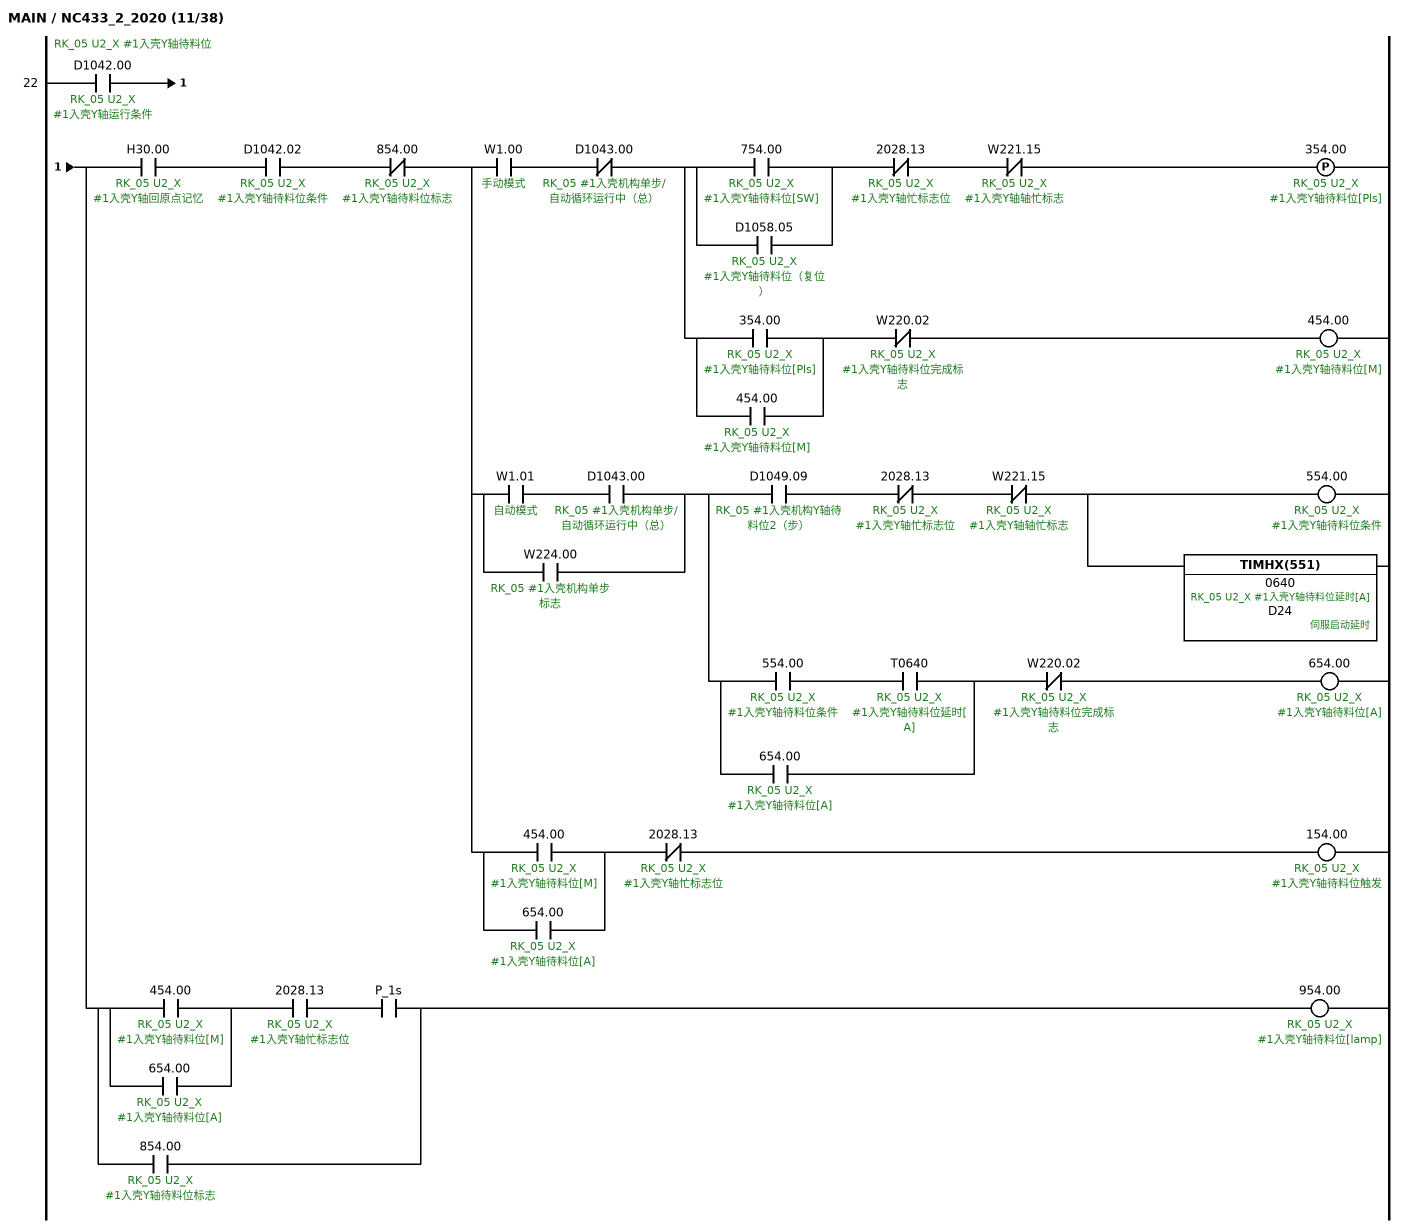
; [picture p120: MAIN / NC433_2_2020, rungs 22-22]
; rung 22: RK_05 U2_X #1入壳Y轴待料位
LD D1042.00  ; RK_05 U2_X #1入壳Y轴运行条件
OUT TR0
AND H30.00  ; RK_05 U2_X #1入壳Y轴回原点记忆
AND D1042.02  ; RK_05 U2_X #1入壳Y轴待料位条件
ANDNOT 854.00  ; RK_05 U2_X #1入壳Y轴待料位标志
OUT TR1
AND W1.00  ; 手动模式
ANDNOT D1043.00  ; RK_05 #1入壳机构单步/自动循环运行中（总）
OUT TR2
LD 754.00  ; RK_05 U2_X #1入壳Y轴待料位[SW]
OR D1058.05  ; RK_05 U2_X #1入壳Y轴待料位（复位）
ANDLD
ANDNOT 2028.13  ; RK_05 U2_X #1入壳Y轴忙标志位
ANDNOT W221.15  ; RK_05 U2_X #1入壳Y轴轴忙标志
DIFU(013) 354.00  ; RK_05 U2_X #1入壳Y轴待料位[Pls]
LD TR2
LD 354.00  ; RK_05 U2_X #1入壳Y轴待料位[Pls]
OR 454.00  ; RK_05 U2_X #1入壳Y轴待料位[M]
ANDLD
ANDNOT W220.02  ; RK_05 U2_X #1入壳Y轴待料位完成标志
OUT 454.00  ; RK_05 U2_X #1入壳Y轴待料位[M]
LD TR1
LD W1.01  ; 自动模式
AND D1043.00  ; RK_05 #1入壳机构单步/自动循环运行中（总）
OR W224.00  ; RK_05 #1入壳机构单步标志
ANDLD
OUT TR2
AND D1049.09  ; RK_05 #1入壳机构Y轴待料位2（步）
ANDNOT 2028.13  ; RK_05 U2_X #1入壳Y轴忙标志位
ANDNOT W221.15  ; RK_05 U2_X #1入壳Y轴轴忙标志
OUT 554.00  ; RK_05 U2_X #1入壳Y轴待料位条件
TIMHX(551) 0640 D24  ; 伺服启动延时, RK_05 U2_X #1入壳Y轴待料位延时[A]
LD TR2
LD 554.00  ; RK_05 U2_X #1入壳Y轴待料位条件
AND T0640  ; RK_05 U2_X #1入壳Y轴待料位延时[A]
OR 654.00  ; RK_05 U2_X #1入壳Y轴待料位[A]
ANDLD
ANDNOT W220.02  ; RK_05 U2_X #1入壳Y轴待料位完成标志
OUT 654.00  ; RK_05 U2_X #1入壳Y轴待料位[A]
LD TR1
LD 454.00  ; RK_05 U2_X #1入壳Y轴待料位[M]
OR 654.00  ; RK_05 U2_X #1入壳Y轴待料位[A]
ANDLD
ANDNOT 2028.13  ; RK_05 U2_X #1入壳Y轴忙标志位
OUT 154.00  ; RK_05 U2_X #1入壳Y轴待料位触发
LD TR0
LD 454.00  ; RK_05 U2_X #1入壳Y轴待料位[M]
OR 654.00  ; RK_05 U2_X #1入壳Y轴待料位[A]
AND 2028.13  ; RK_05 U2_X #1入壳Y轴忙标志位
AND P_1s
OR 854.00  ; RK_05 U2_X #1入壳Y轴待料位标志
ANDLD
OUT 954.00  ; RK_05 U2_X #1入壳Y轴待料位[lamp]

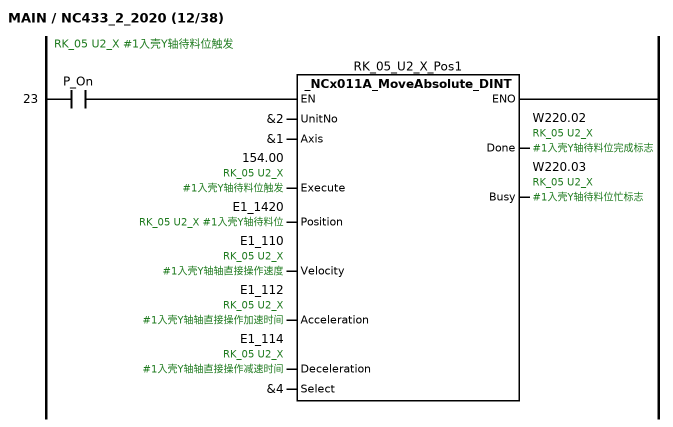
; rung 23: RK_05 U2_X #1入壳Y轴待料位触发
LD P_On
CALL RK_05_U2_X_Pos1 : _NCx011A_MoveAbsolute_DINT (UnitNo := &2, Axis := &1, Execute := 154.00, Position := E1_1420, Velocity := E1_110, Acceleration := E1_112, Deceleration := E1_114, Select := &4, Done => W220.02, Busy => W220.03)  ; RK_05 U2_X #1入壳Y轴待料位触发, RK_05 U2_X #1入壳Y轴待料位, RK_05 U2_X #1入壳Y轴轴直接操作速度, RK_05 U2_X #1入壳Y轴轴直接操作加速时间, RK_05 U2_X #1入壳Y轴轴直接操作减速时间, RK_05 U2_X #1入壳Y轴待料位完成标志, RK_05 U2_X #1入壳Y轴待料位忙标志

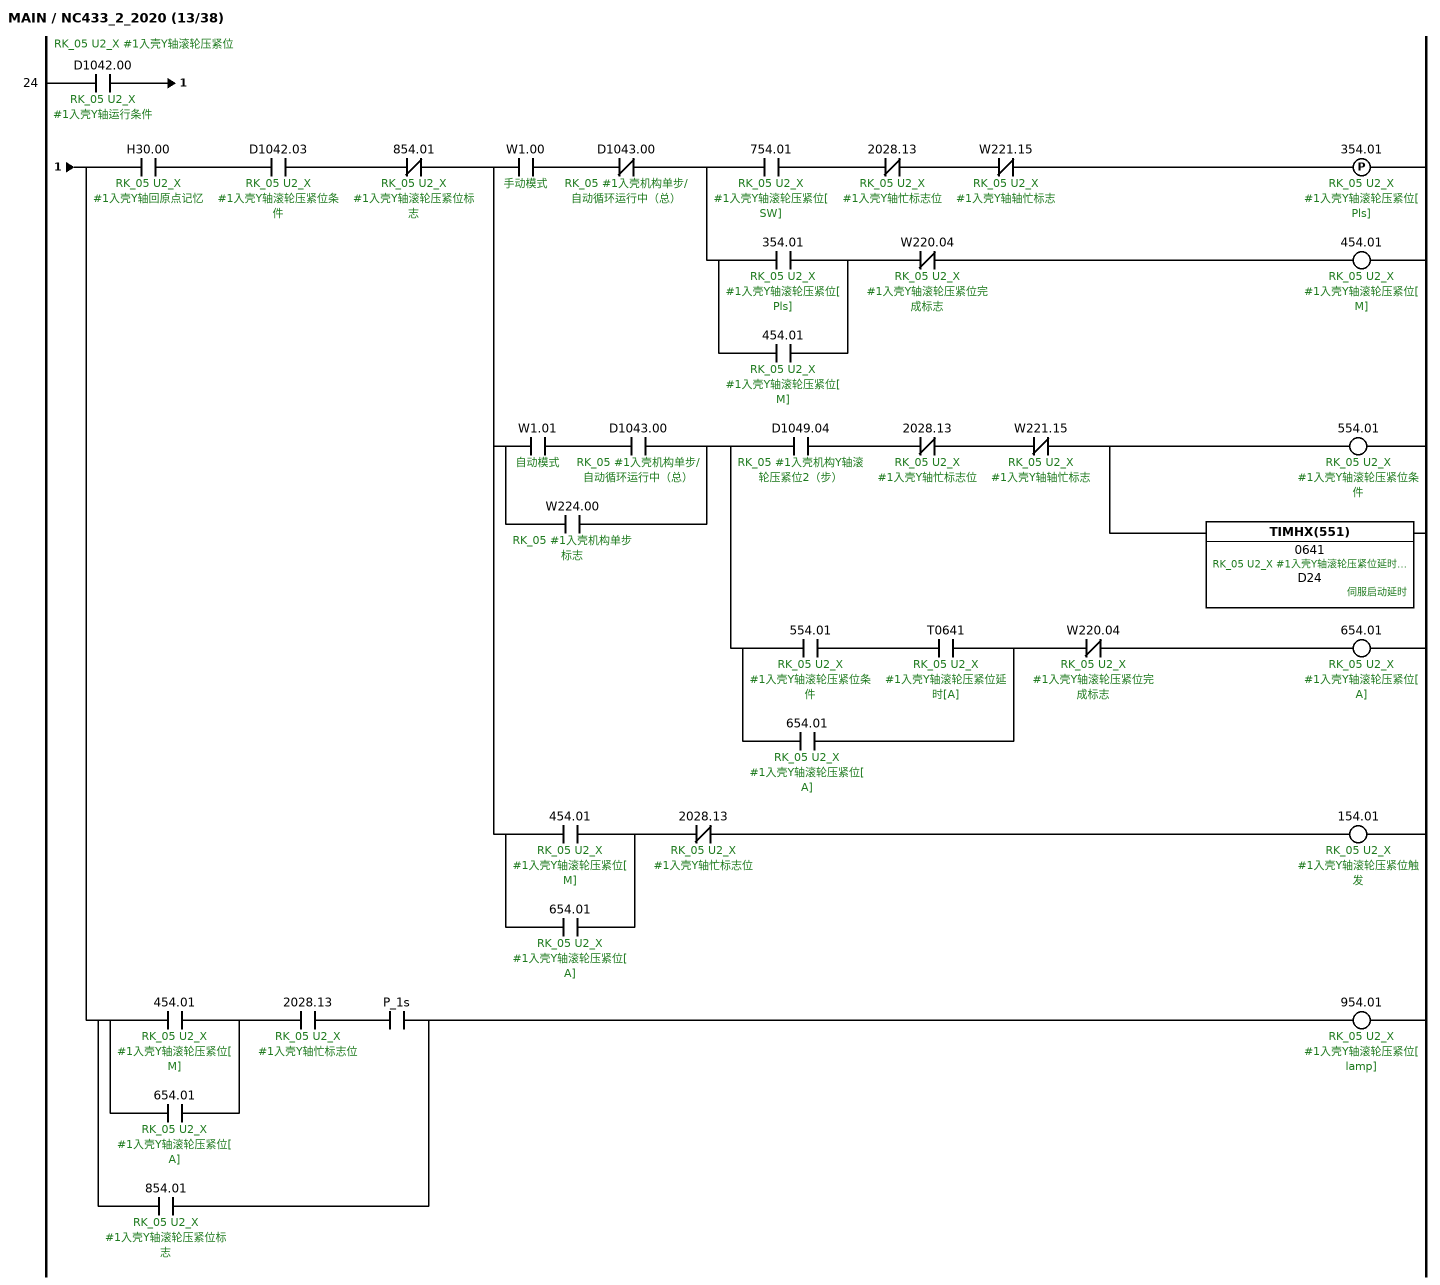
; rung 24: RK_05 U2_X #1入壳Y轴滚轮压紧位
LD D1042.00  ; RK_05 U2_X #1入壳Y轴运行条件
OUT TR0
AND H30.00  ; RK_05 U2_X #1入壳Y轴回原点记忆
AND D1042.03  ; RK_05 U2_X #1入壳Y轴滚轮压紧位条件
ANDNOT 854.01  ; RK_05 U2_X #1入壳Y轴滚轮压紧位标志
OUT TR1
AND W1.00  ; 手动模式
ANDNOT D1043.00  ; RK_05 #1入壳机构单步/自动循环运行中（总）
OUT TR2
AND 754.01  ; RK_05 U2_X #1入壳Y轴滚轮压紧位[SW]
ANDNOT 2028.13  ; RK_05 U2_X #1入壳Y轴忙标志位
ANDNOT W221.15  ; RK_05 U2_X #1入壳Y轴轴忙标志
DIFU(013) 354.01  ; RK_05 U2_X #1入壳Y轴滚轮压紧位[Pls]
LD TR2
LD 354.01  ; RK_05 U2_X #1入壳Y轴滚轮压紧位[Pls]
OR 454.01  ; RK_05 U2_X #1入壳Y轴滚轮压紧位[M]
ANDLD
ANDNOT W220.04  ; RK_05 U2_X #1入壳Y轴滚轮压紧位完成标志
OUT 454.01  ; RK_05 U2_X #1入壳Y轴滚轮压紧位[M]
LD TR1
LD W1.01  ; 自动模式
AND D1043.00  ; RK_05 #1入壳机构单步/自动循环运行中（总）
OR W224.00  ; RK_05 #1入壳机构单步标志
ANDLD
OUT TR2
AND D1049.04  ; RK_05 #1入壳机构Y轴滚轮压紧位2（步）
ANDNOT 2028.13  ; RK_05 U2_X #1入壳Y轴忙标志位
ANDNOT W221.15  ; RK_05 U2_X #1入壳Y轴轴忙标志
OUT 554.01  ; RK_05 U2_X #1入壳Y轴滚轮压紧位条件
TIMHX(551) 0641 D24  ; 伺服启动延时, RK_05 U2_X #1入壳Y轴滚轮压紧位延时[A]
LD TR2
LD 554.01  ; RK_05 U2_X #1入壳Y轴滚轮压紧位条件
AND T0641  ; RK_05 U2_X #1入壳Y轴滚轮压紧位延时[A]
OR 654.01  ; RK_05 U2_X #1入壳Y轴滚轮压紧位[A]
ANDLD
ANDNOT W220.04  ; RK_05 U2_X #1入壳Y轴滚轮压紧位完成标志
OUT 654.01  ; RK_05 U2_X #1入壳Y轴滚轮压紧位[A]
LD TR1
LD 454.01  ; RK_05 U2_X #1入壳Y轴滚轮压紧位[M]
OR 654.01  ; RK_05 U2_X #1入壳Y轴滚轮压紧位[A]
ANDLD
ANDNOT 2028.13  ; RK_05 U2_X #1入壳Y轴忙标志位
OUT 154.01  ; RK_05 U2_X #1入壳Y轴滚轮压紧位触发
LD TR0
LD 454.01  ; RK_05 U2_X #1入壳Y轴滚轮压紧位[M]
OR 654.01  ; RK_05 U2_X #1入壳Y轴滚轮压紧位[A]
AND 2028.13  ; RK_05 U2_X #1入壳Y轴忙标志位
AND P_1s
OR 854.01  ; RK_05 U2_X #1入壳Y轴滚轮压紧位标志
ANDLD
OUT 954.01  ; RK_05 U2_X #1入壳Y轴滚轮压紧位[lamp]

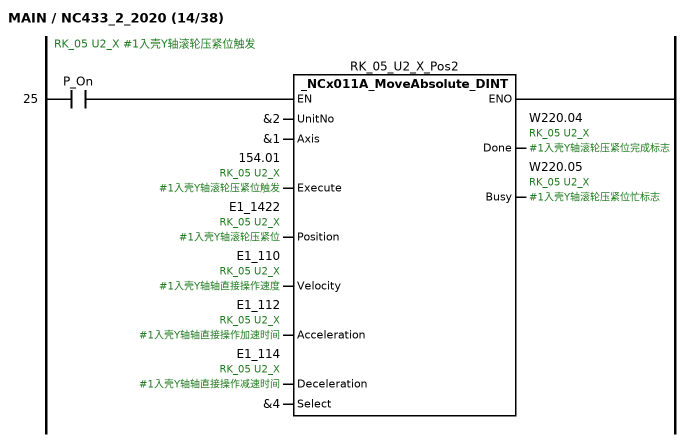
; rung 25: RK_05 U2_X #1入壳Y轴滚轮压紧位触发
LD P_On
CALL RK_05_U2_X_Pos2 : _NCx011A_MoveAbsolute_DINT (UnitNo := &2, Axis := &1, Execute := 154.01, Position := E1_1422, Velocity := E1_110, Acceleration := E1_112, Deceleration := E1_114, Select := &4, Done => W220.04, Busy => W220.05)  ; RK_05 U2_X #1入壳Y轴滚轮压紧位触发, RK_05 U2_X #1入壳Y轴滚轮压紧位, RK_05 U2_X #1入壳Y轴轴直接操作速度, RK_05 U2_X #1入壳Y轴轴直接操作加速时间, RK_05 U2_X #1入壳Y轴轴直接操作减速时间, RK_05 U2_X #1入壳Y轴滚轮压紧位完成标志, RK_05 U2_X #1入壳Y轴滚轮压紧位忙标志

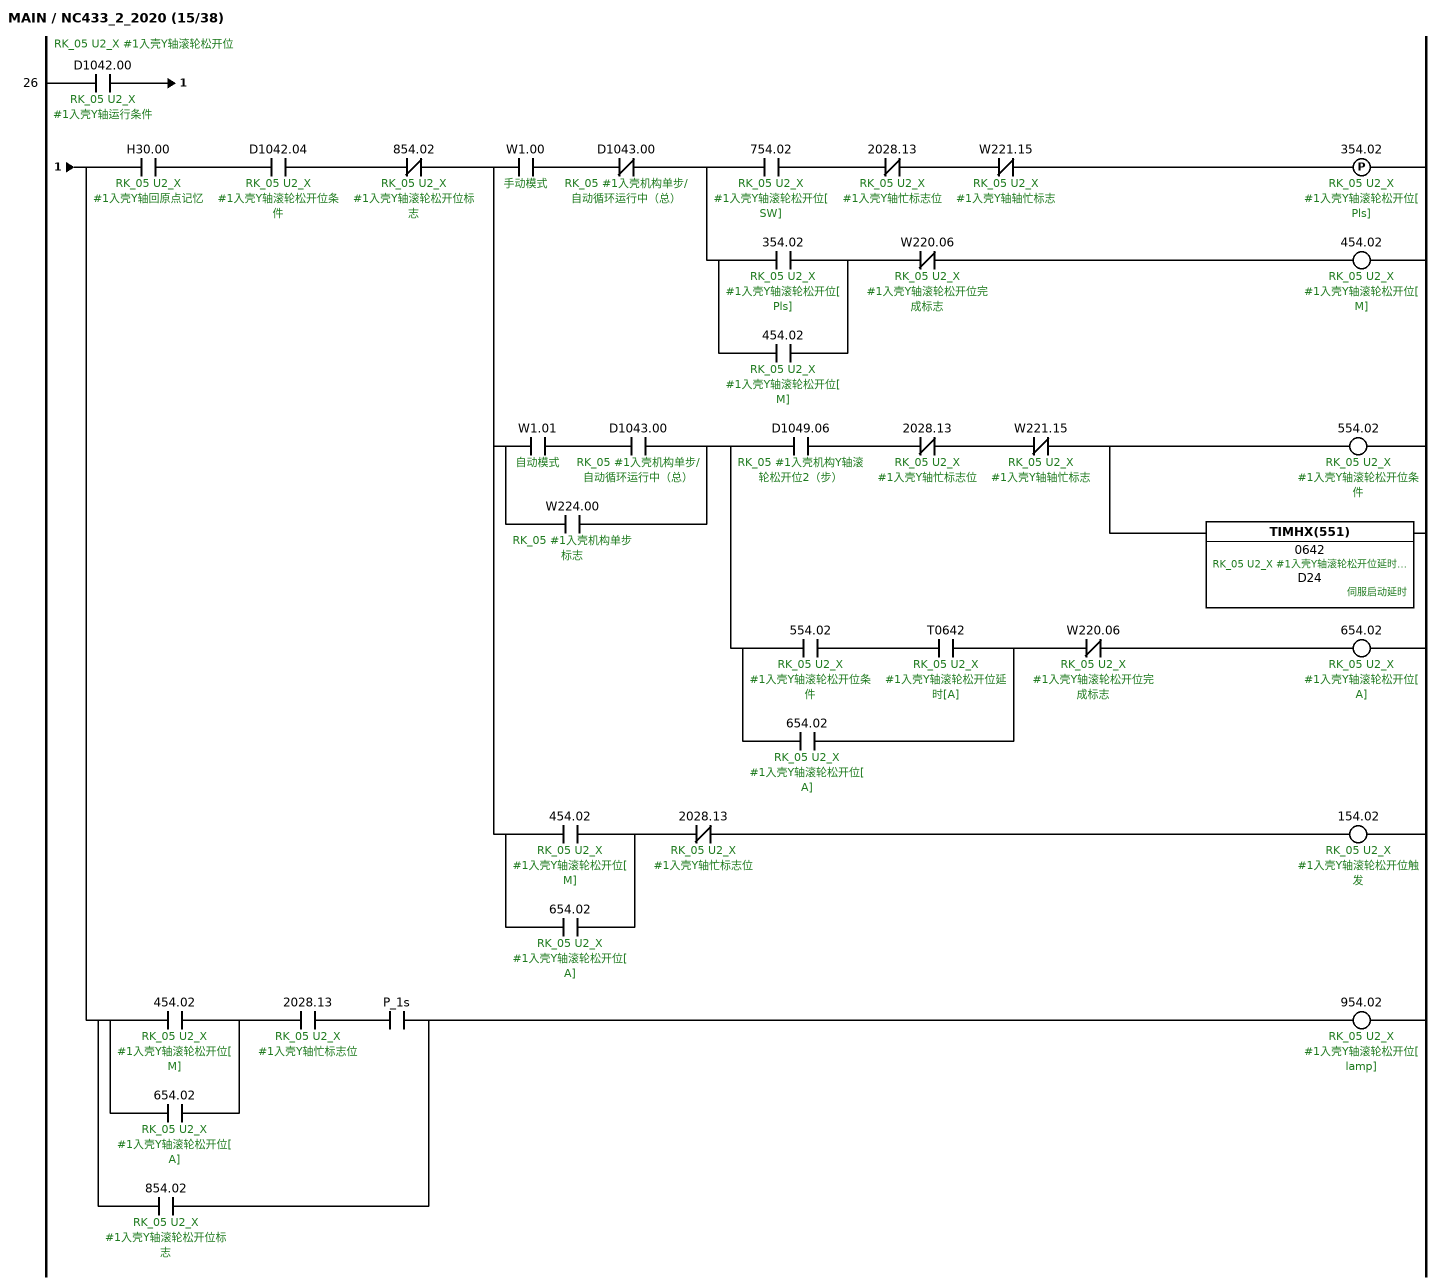
; rung 26: RK_05 U2_X #1入壳Y轴滚轮松开位
LD D1042.00  ; RK_05 U2_X #1入壳Y轴运行条件
OUT TR0
AND H30.00  ; RK_05 U2_X #1入壳Y轴回原点记忆
AND D1042.04  ; RK_05 U2_X #1入壳Y轴滚轮松开位条件
ANDNOT 854.02  ; RK_05 U2_X #1入壳Y轴滚轮松开位标志
OUT TR1
AND W1.00  ; 手动模式
ANDNOT D1043.00  ; RK_05 #1入壳机构单步/自动循环运行中（总）
OUT TR2
AND 754.02  ; RK_05 U2_X #1入壳Y轴滚轮松开位[SW]
ANDNOT 2028.13  ; RK_05 U2_X #1入壳Y轴忙标志位
ANDNOT W221.15  ; RK_05 U2_X #1入壳Y轴轴忙标志
DIFU(013) 354.02  ; RK_05 U2_X #1入壳Y轴滚轮松开位[Pls]
LD TR2
LD 354.02  ; RK_05 U2_X #1入壳Y轴滚轮松开位[Pls]
OR 454.02  ; RK_05 U2_X #1入壳Y轴滚轮松开位[M]
ANDLD
ANDNOT W220.06  ; RK_05 U2_X #1入壳Y轴滚轮松开位完成标志
OUT 454.02  ; RK_05 U2_X #1入壳Y轴滚轮松开位[M]
LD TR1
LD W1.01  ; 自动模式
AND D1043.00  ; RK_05 #1入壳机构单步/自动循环运行中（总）
OR W224.00  ; RK_05 #1入壳机构单步标志
ANDLD
OUT TR2
AND D1049.06  ; RK_05 #1入壳机构Y轴滚轮松开位2（步）
ANDNOT 2028.13  ; RK_05 U2_X #1入壳Y轴忙标志位
ANDNOT W221.15  ; RK_05 U2_X #1入壳Y轴轴忙标志
OUT 554.02  ; RK_05 U2_X #1入壳Y轴滚轮松开位条件
TIMHX(551) 0642 D24  ; 伺服启动延时, RK_05 U2_X #1入壳Y轴滚轮松开位延时[A]
LD TR2
LD 554.02  ; RK_05 U2_X #1入壳Y轴滚轮松开位条件
AND T0642  ; RK_05 U2_X #1入壳Y轴滚轮松开位延时[A]
OR 654.02  ; RK_05 U2_X #1入壳Y轴滚轮松开位[A]
ANDLD
ANDNOT W220.06  ; RK_05 U2_X #1入壳Y轴滚轮松开位完成标志
OUT 654.02  ; RK_05 U2_X #1入壳Y轴滚轮松开位[A]
LD TR1
LD 454.02  ; RK_05 U2_X #1入壳Y轴滚轮松开位[M]
OR 654.02  ; RK_05 U2_X #1入壳Y轴滚轮松开位[A]
ANDLD
ANDNOT 2028.13  ; RK_05 U2_X #1入壳Y轴忙标志位
OUT 154.02  ; RK_05 U2_X #1入壳Y轴滚轮松开位触发
LD TR0
LD 454.02  ; RK_05 U2_X #1入壳Y轴滚轮松开位[M]
OR 654.02  ; RK_05 U2_X #1入壳Y轴滚轮松开位[A]
AND 2028.13  ; RK_05 U2_X #1入壳Y轴忙标志位
AND P_1s
OR 854.02  ; RK_05 U2_X #1入壳Y轴滚轮松开位标志
ANDLD
OUT 954.02  ; RK_05 U2_X #1入壳Y轴滚轮松开位[lamp]

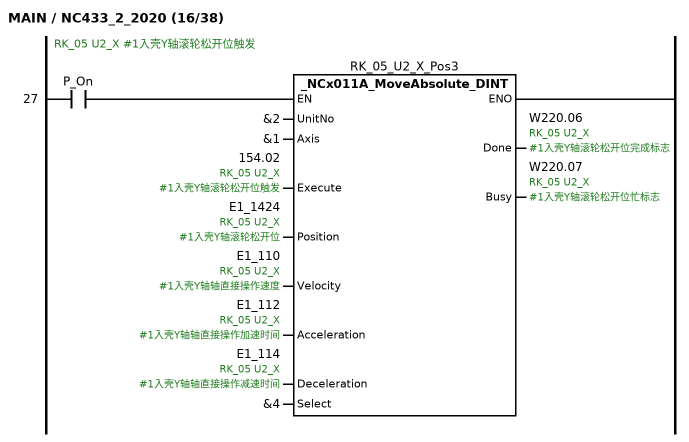
; rung 27: RK_05 U2_X #1入壳Y轴滚轮松开位触发
LD P_On
CALL RK_05_U2_X_Pos3 : _NCx011A_MoveAbsolute_DINT (UnitNo := &2, Axis := &1, Execute := 154.02, Position := E1_1424, Velocity := E1_110, Acceleration := E1_112, Deceleration := E1_114, Select := &4, Done => W220.06, Busy => W220.07)  ; RK_05 U2_X #1入壳Y轴滚轮松开位触发, RK_05 U2_X #1入壳Y轴滚轮松开位, RK_05 U2_X #1入壳Y轴轴直接操作速度, RK_05 U2_X #1入壳Y轴轴直接操作加速时间, RK_05 U2_X #1入壳Y轴轴直接操作减速时间, RK_05 U2_X #1入壳Y轴滚轮松开位完成标志, RK_05 U2_X #1入壳Y轴滚轮松开位忙标志

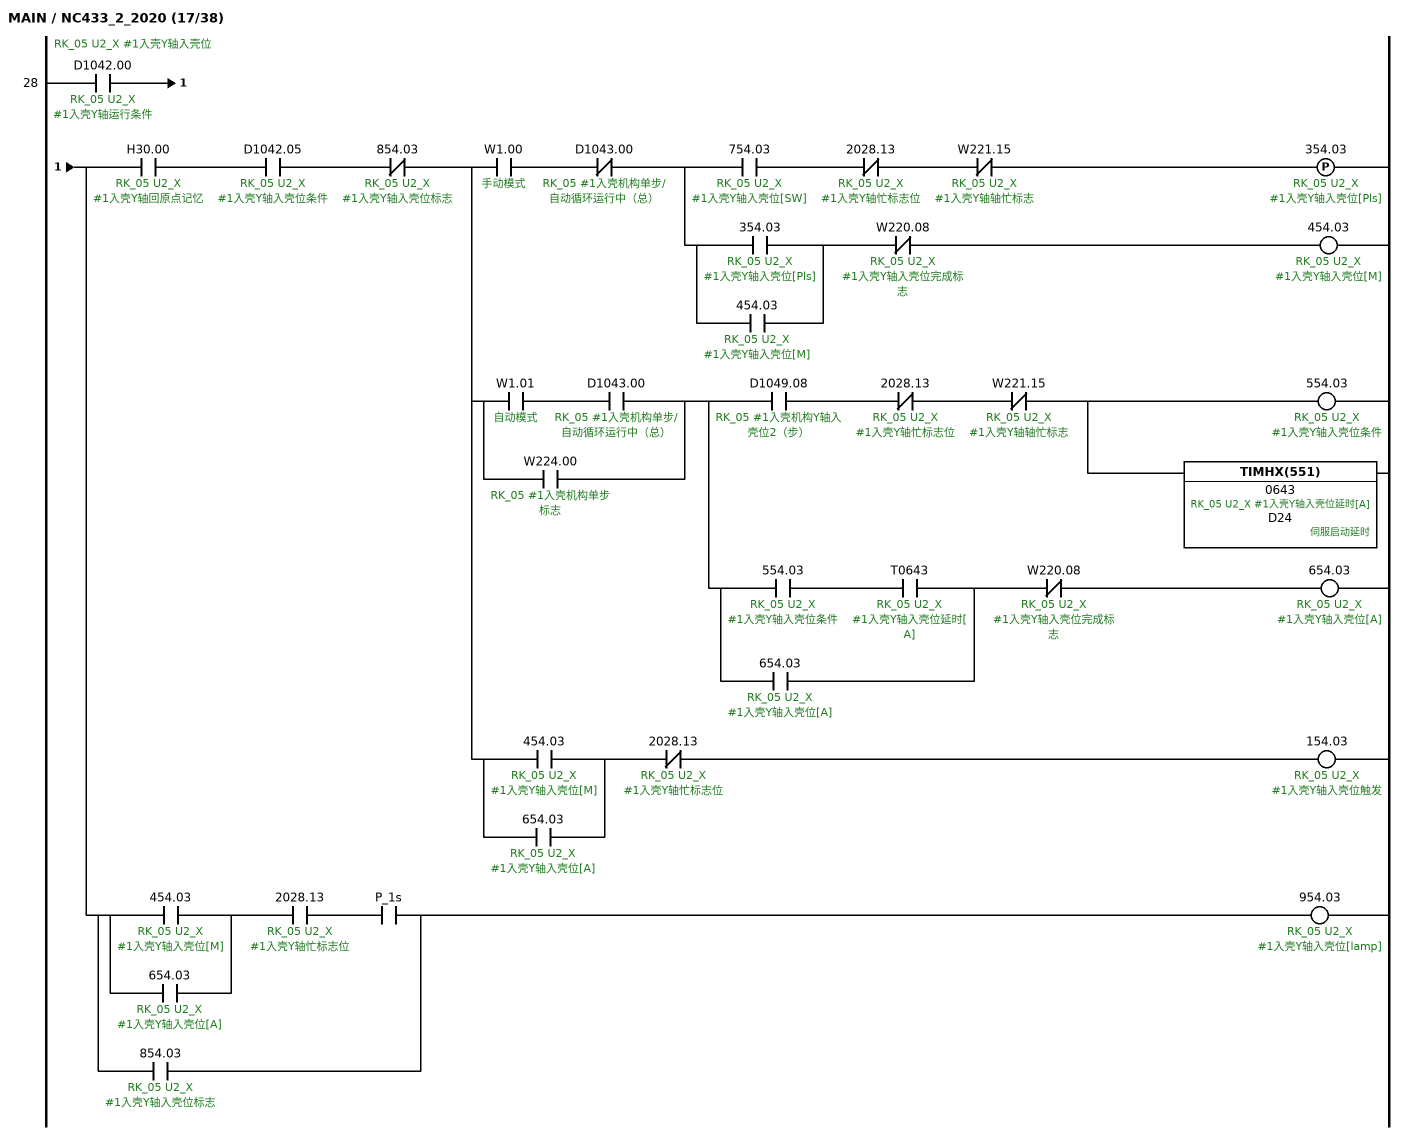
; rung 28: RK_05 U2_X #1入壳Y轴入壳位
LD D1042.00  ; RK_05 U2_X #1入壳Y轴运行条件
OUT TR0
AND H30.00  ; RK_05 U2_X #1入壳Y轴回原点记忆
AND D1042.05  ; RK_05 U2_X #1入壳Y轴入壳位条件
ANDNOT 854.03  ; RK_05 U2_X #1入壳Y轴入壳位标志
OUT TR1
AND W1.00  ; 手动模式
ANDNOT D1043.00  ; RK_05 #1入壳机构单步/自动循环运行中（总）
OUT TR2
AND 754.03  ; RK_05 U2_X #1入壳Y轴入壳位[SW]
ANDNOT 2028.13  ; RK_05 U2_X #1入壳Y轴忙标志位
ANDNOT W221.15  ; RK_05 U2_X #1入壳Y轴轴忙标志
DIFU(013) 354.03  ; RK_05 U2_X #1入壳Y轴入壳位[Pls]
LD TR2
LD 354.03  ; RK_05 U2_X #1入壳Y轴入壳位[Pls]
OR 454.03  ; RK_05 U2_X #1入壳Y轴入壳位[M]
ANDLD
ANDNOT W220.08  ; RK_05 U2_X #1入壳Y轴入壳位完成标志
OUT 454.03  ; RK_05 U2_X #1入壳Y轴入壳位[M]
LD TR1
LD W1.01  ; 自动模式
AND D1043.00  ; RK_05 #1入壳机构单步/自动循环运行中（总）
OR W224.00  ; RK_05 #1入壳机构单步标志
ANDLD
OUT TR2
AND D1049.08  ; RK_05 #1入壳机构Y轴入壳位2（步）
ANDNOT 2028.13  ; RK_05 U2_X #1入壳Y轴忙标志位
ANDNOT W221.15  ; RK_05 U2_X #1入壳Y轴轴忙标志
OUT 554.03  ; RK_05 U2_X #1入壳Y轴入壳位条件
TIMHX(551) 0643 D24  ; 伺服启动延时, RK_05 U2_X #1入壳Y轴入壳位延时[A]
LD TR2
LD 554.03  ; RK_05 U2_X #1入壳Y轴入壳位条件
AND T0643  ; RK_05 U2_X #1入壳Y轴入壳位延时[A]
OR 654.03  ; RK_05 U2_X #1入壳Y轴入壳位[A]
ANDLD
ANDNOT W220.08  ; RK_05 U2_X #1入壳Y轴入壳位完成标志
OUT 654.03  ; RK_05 U2_X #1入壳Y轴入壳位[A]
LD TR1
LD 454.03  ; RK_05 U2_X #1入壳Y轴入壳位[M]
OR 654.03  ; RK_05 U2_X #1入壳Y轴入壳位[A]
ANDLD
ANDNOT 2028.13  ; RK_05 U2_X #1入壳Y轴忙标志位
OUT 154.03  ; RK_05 U2_X #1入壳Y轴入壳位触发
LD TR0
LD 454.03  ; RK_05 U2_X #1入壳Y轴入壳位[M]
OR 654.03  ; RK_05 U2_X #1入壳Y轴入壳位[A]
AND 2028.13  ; RK_05 U2_X #1入壳Y轴忙标志位
AND P_1s
OR 854.03  ; RK_05 U2_X #1入壳Y轴入壳位标志
ANDLD
OUT 954.03  ; RK_05 U2_X #1入壳Y轴入壳位[lamp]

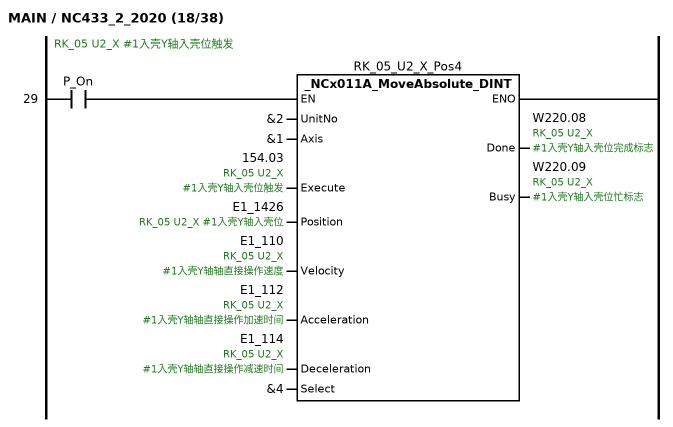
; rung 29: RK_05 U2_X #1入壳Y轴入壳位触发
LD P_On
CALL RK_05_U2_X_Pos4 : _NCx011A_MoveAbsolute_DINT (UnitNo := &2, Axis := &1, Execute := 154.03, Position := E1_1426, Velocity := E1_110, Acceleration := E1_112, Deceleration := E1_114, Select := &4, Done => W220.08, Busy => W220.09)  ; RK_05 U2_X #1入壳Y轴入壳位触发, RK_05 U2_X #1入壳Y轴入壳位, RK_05 U2_X #1入壳Y轴轴直接操作速度, RK_05 U2_X #1入壳Y轴轴直接操作加速时间, RK_05 U2_X #1入壳Y轴轴直接操作减速时间, RK_05 U2_X #1入壳Y轴入壳位完成标志, RK_05 U2_X #1入壳Y轴入壳位忙标志

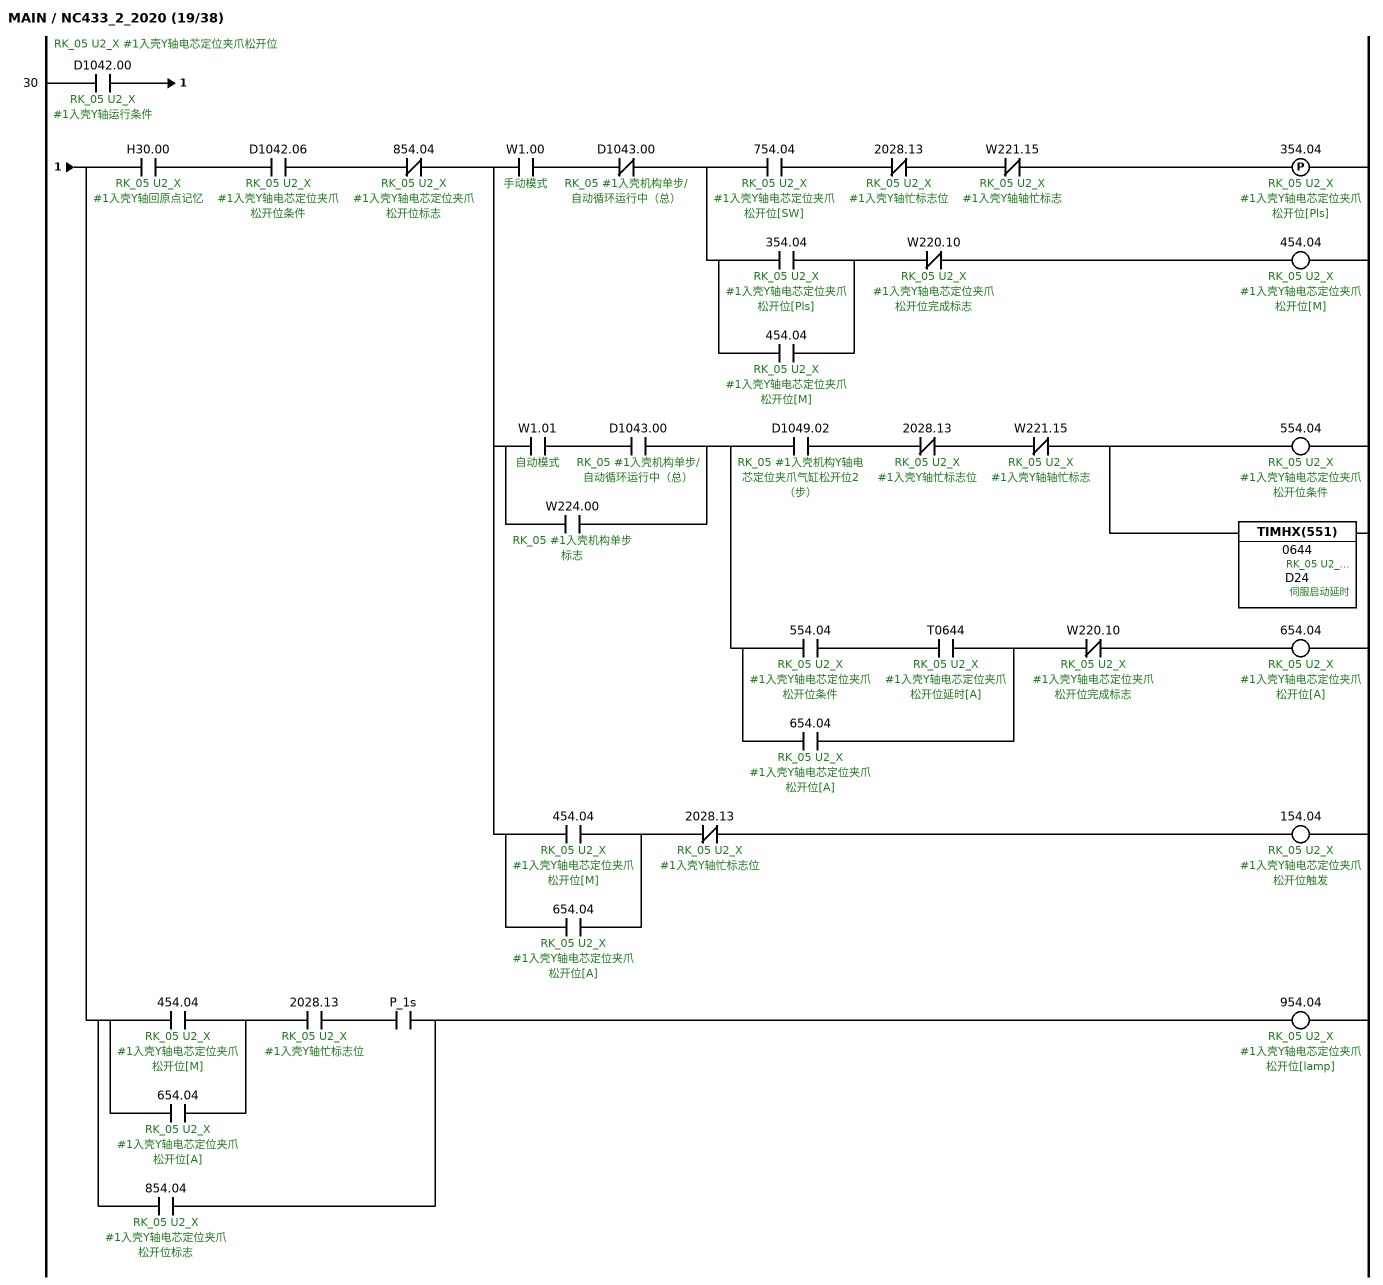
; rung 30: RK_05 U2_X #1入壳Y轴电芯定位夹爪松开位
LD D1042.00  ; RK_05 U2_X #1入壳Y轴运行条件
OUT TR0
AND H30.00  ; RK_05 U2_X #1入壳Y轴回原点记忆
AND D1042.06  ; RK_05 U2_X #1入壳Y轴电芯定位夹爪松开位条件
ANDNOT 854.04  ; RK_05 U2_X #1入壳Y轴电芯定位夹爪松开位标志
OUT TR1
AND W1.00  ; 手动模式
ANDNOT D1043.00  ; RK_05 #1入壳机构单步/自动循环运行中（总）
OUT TR2
AND 754.04  ; RK_05 U2_X #1入壳Y轴电芯定位夹爪松开位[SW]
ANDNOT 2028.13  ; RK_05 U2_X #1入壳Y轴忙标志位
ANDNOT W221.15  ; RK_05 U2_X #1入壳Y轴轴忙标志
DIFU(013) 354.04  ; RK_05 U2_X #1入壳Y轴电芯定位夹爪松开位[Pls]
LD TR2
LD 354.04  ; RK_05 U2_X #1入壳Y轴电芯定位夹爪松开位[Pls]
OR 454.04  ; RK_05 U2_X #1入壳Y轴电芯定位夹爪松开位[M]
ANDLD
ANDNOT W220.10  ; RK_05 U2_X #1入壳Y轴电芯定位夹爪松开位完成标志
OUT 454.04  ; RK_05 U2_X #1入壳Y轴电芯定位夹爪松开位[M]
LD TR1
LD W1.01  ; 自动模式
AND D1043.00  ; RK_05 #1入壳机构单步/自动循环运行中（总）
OR W224.00  ; RK_05 #1入壳机构单步标志
ANDLD
OUT TR2
AND D1049.02  ; RK_05 #1入壳机构Y轴电芯定位夹爪气缸松开位2（步）
ANDNOT 2028.13  ; RK_05 U2_X #1入壳Y轴忙标志位
ANDNOT W221.15  ; RK_05 U2_X #1入壳Y轴轴忙标志
OUT 554.04  ; RK_05 U2_X #1入壳Y轴电芯定位夹爪松开位条件
TIMHX(551) 0644 D24  ; 伺服启动延时, RK_05 U2_X #1入壳Y轴电芯定位夹爪松开位延时[A]
LD TR2
LD 554.04  ; RK_05 U2_X #1入壳Y轴电芯定位夹爪松开位条件
AND T0644  ; RK_05 U2_X #1入壳Y轴电芯定位夹爪松开位延时[A]
OR 654.04  ; RK_05 U2_X #1入壳Y轴电芯定位夹爪松开位[A]
ANDLD
ANDNOT W220.10  ; RK_05 U2_X #1入壳Y轴电芯定位夹爪松开位完成标志
OUT 654.04  ; RK_05 U2_X #1入壳Y轴电芯定位夹爪松开位[A]
LD TR1
LD 454.04  ; RK_05 U2_X #1入壳Y轴电芯定位夹爪松开位[M]
OR 654.04  ; RK_05 U2_X #1入壳Y轴电芯定位夹爪松开位[A]
ANDLD
ANDNOT 2028.13  ; RK_05 U2_X #1入壳Y轴忙标志位
OUT 154.04  ; RK_05 U2_X #1入壳Y轴电芯定位夹爪松开位触发
LD TR0
LD 454.04  ; RK_05 U2_X #1入壳Y轴电芯定位夹爪松开位[M]
OR 654.04  ; RK_05 U2_X #1入壳Y轴电芯定位夹爪松开位[A]
AND 2028.13  ; RK_05 U2_X #1入壳Y轴忙标志位
AND P_1s
OR 854.04  ; RK_05 U2_X #1入壳Y轴电芯定位夹爪松开位标志
ANDLD
OUT 954.04  ; RK_05 U2_X #1入壳Y轴电芯定位夹爪松开位[lamp]

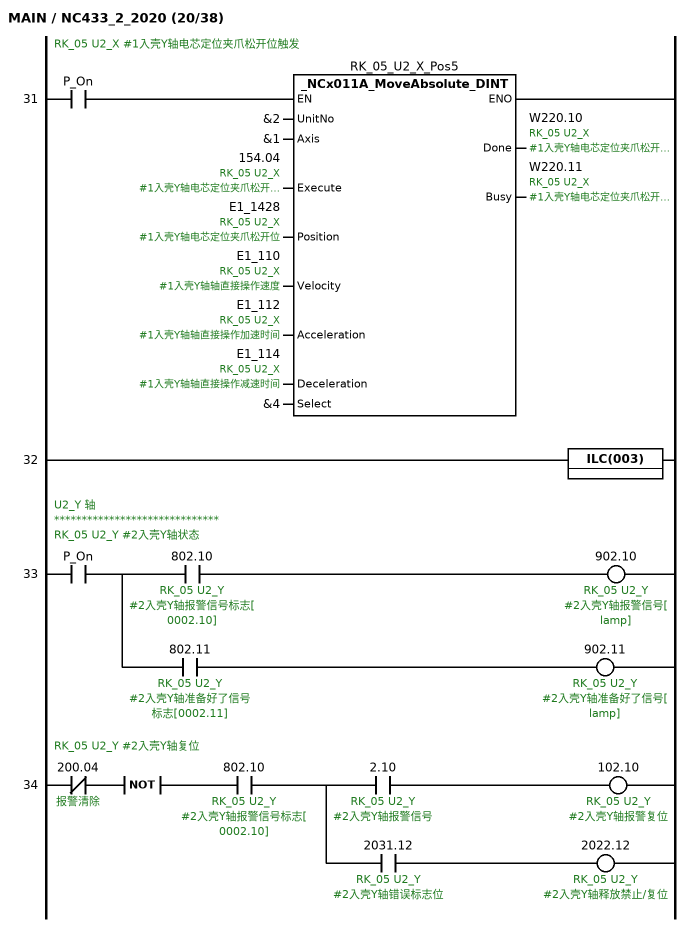
; rung 31: RK_05 U2_X #1入壳Y轴电芯定位夹爪松开位触发
LD P_On
CALL RK_05_U2_X_Pos5 : _NCx011A_MoveAbsolute_DINT (UnitNo := &2, Axis := &1, Execute := 154.04, Position := E1_1428, Velocity := E1_110, Acceleration := E1_112, Deceleration := E1_114, Select := &4, Done => W220.10, Busy => W220.11)  ; RK_05 U2_X #1入壳Y轴电芯定位夹爪松开位触发, RK_05 U2_X #1入壳Y轴电芯定位夹爪松开位, RK_05 U2_X #1入壳Y轴轴直接操作速度, RK_05 U2_X #1入壳Y轴轴直接操作加速时间, RK_05 U2_X #1入壳Y轴轴直接操作减速时间, RK_05 U2_X #1入壳Y轴电芯定位夹爪松开位完成标志, RK_05 U2_X #1入壳Y轴电芯定位夹爪松开位忙标志
; rung 32
ILC(003)
; rung 33: U2_Y 轴 / ****************************** / RK_05 U2_Y #2入壳Y轴状态
LD P_On
OUT TR0
AND 802.10  ; RK_05 U2_Y #2入壳Y轴报警信号标志[0002.10]
OUT 902.10  ; RK_05 U2_Y #2入壳Y轴报警信号[lamp]
LD TR0
AND 802.11  ; RK_05 U2_Y #2入壳Y轴准备好了信号标志[0002.11]
OUT 902.11  ; RK_05 U2_Y #2入壳Y轴准备好了信号[lamp]
; rung 34: RK_05 U2_Y #2入壳Y轴复位
LDNOT 200.04  ; 报警清除
NOT(520)
AND 802.10  ; RK_05 U2_Y #2入壳Y轴报警信号标志[0002.10]
OUT TR0
AND 2.10  ; RK_05 U2_Y #2入壳Y轴报警信号
OUT 102.10  ; RK_05 U2_Y #2入壳Y轴报警复位
LD TR0
AND 2031.12  ; RK_05 U2_Y #2入壳Y轴错误标志位
OUT 2022.12  ; RK_05 U2_Y #2入壳Y轴释放禁止/复位

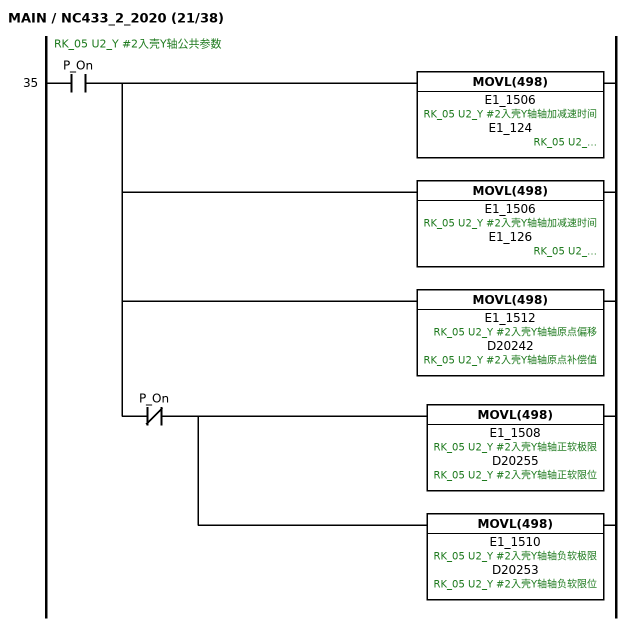
; rung 35: RK_05 U2_Y #2入壳Y轴公共参数
LD P_On
MOVL(498) E1_1506 E1_124  ; RK_05 U2_Y #2入壳Y轴轴加减速时间, RK_05 U2_Y #2入壳Y轴轴直接操作加速时间
MOVL(498) E1_1506 E1_126  ; RK_05 U2_Y #2入壳Y轴轴加减速时间, RK_05 U2_Y #2入壳Y轴轴直接操作减速时间
MOVL(498) E1_1512 D20242  ; RK_05 U2_Y #2入壳Y轴轴原点偏移, RK_05 U2_Y #2入壳Y轴轴原点补偿值
ANDNOT P_On
MOVL(498) E1_1508 D20255  ; RK_05 U2_Y #2入壳Y轴轴正软极限, RK_05 U2_Y #2入壳Y轴轴正软限位
MOVL(498) E1_1510 D20253  ; RK_05 U2_Y #2入壳Y轴轴负软极限, RK_05 U2_Y #2入壳Y轴轴负软限位

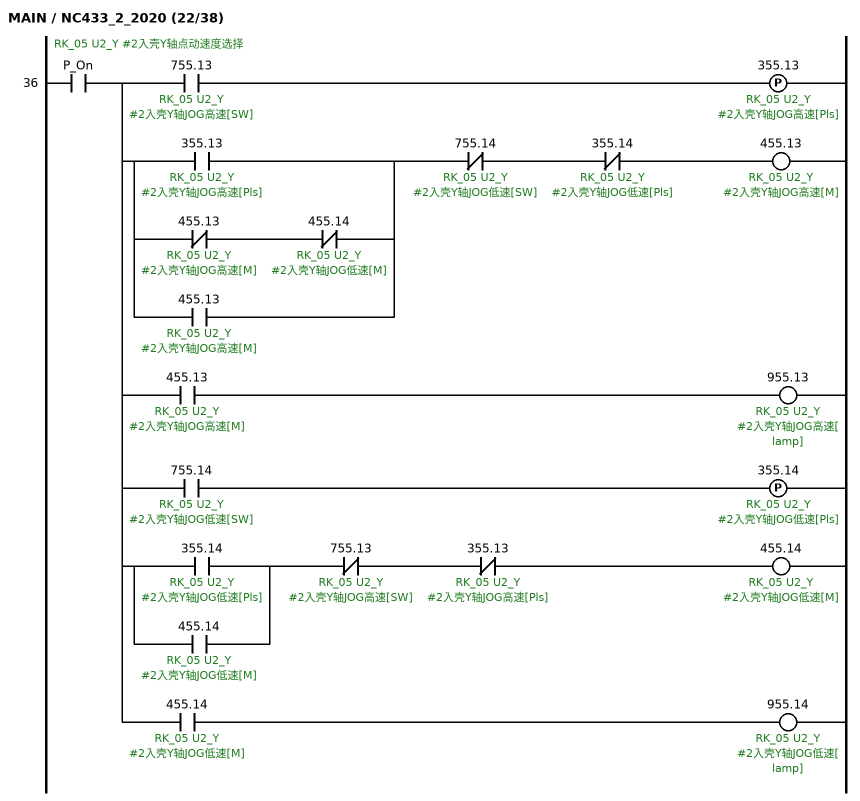
; rung 36: RK_05 U2_Y #2入壳Y轴点动速度选择
LD P_On
OUT TR0
AND 755.13  ; RK_05 U2_Y #2入壳Y轴JOG高速[SW]
DIFU(013) 355.13  ; RK_05 U2_Y #2入壳Y轴JOG高速[Pls]
LD TR0
LD 355.13  ; RK_05 U2_Y #2入壳Y轴JOG高速[Pls]
LDNOT 455.13  ; RK_05 U2_Y #2入壳Y轴JOG高速[M]
ANDNOT 455.14  ; RK_05 U2_Y #2入壳Y轴JOG低速[M]
ORLD
OR 455.13  ; RK_05 U2_Y #2入壳Y轴JOG高速[M]
ANDLD
ANDNOT 755.14  ; RK_05 U2_Y #2入壳Y轴JOG低速[SW]
ANDNOT 355.14  ; RK_05 U2_Y #2入壳Y轴JOG低速[Pls]
OUT 455.13  ; RK_05 U2_Y #2入壳Y轴JOG高速[M]
LD TR0
AND 455.13  ; RK_05 U2_Y #2入壳Y轴JOG高速[M]
OUT 955.13  ; RK_05 U2_Y #2入壳Y轴JOG高速[lamp]
LD TR0
AND 755.14  ; RK_05 U2_Y #2入壳Y轴JOG低速[SW]
DIFU(013) 355.14  ; RK_05 U2_Y #2入壳Y轴JOG低速[Pls]
LD TR0
LD 355.14  ; RK_05 U2_Y #2入壳Y轴JOG低速[Pls]
OR 455.14  ; RK_05 U2_Y #2入壳Y轴JOG低速[M]
ANDLD
ANDNOT 755.13  ; RK_05 U2_Y #2入壳Y轴JOG高速[SW]
ANDNOT 355.13  ; RK_05 U2_Y #2入壳Y轴JOG高速[Pls]
OUT 455.14  ; RK_05 U2_Y #2入壳Y轴JOG低速[M]
LD TR0
AND 455.14  ; RK_05 U2_Y #2入壳Y轴JOG低速[M]
OUT 955.14  ; RK_05 U2_Y #2入壳Y轴JOG低速[lamp]

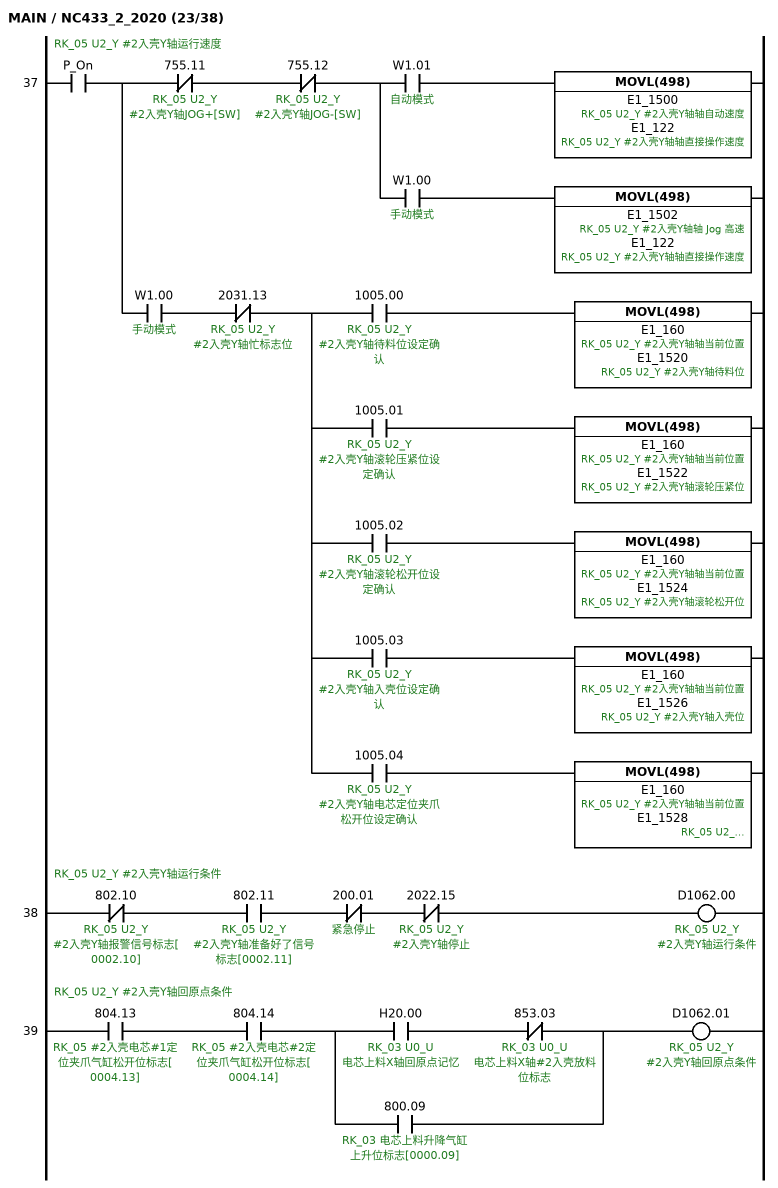
; rung 37: RK_05 U2_Y #2入壳Y轴运行速度
LD P_On
OUT TR0
ANDNOT 755.11  ; RK_05 U2_Y #2入壳Y轴JOG+[SW]
ANDNOT 755.12  ; RK_05 U2_Y #2入壳Y轴JOG-[SW]
OUT TR1
AND W1.01  ; 自动模式
MOVL(498) E1_1500 E1_122  ; RK_05 U2_Y #2入壳Y轴轴自动速度, RK_05 U2_Y #2入壳Y轴轴直接操作速度
LD TR1
AND W1.00  ; 手动模式
MOVL(498) E1_1502 E1_122  ; RK_05 U2_Y #2入壳Y轴轴 Jog 高速, RK_05 U2_Y #2入壳Y轴轴直接操作速度
LD TR0
AND W1.00  ; 手动模式
ANDNOT 2031.13  ; RK_05 U2_Y #2入壳Y轴忙标志位
OUT TR0
AND 1005.00  ; RK_05 U2_Y #2入壳Y轴待料位设定确认
MOVL(498) E1_160 E1_1520  ; RK_05 U2_Y #2入壳Y轴轴当前位置, RK_05 U2_Y #2入壳Y轴待料位
LD TR0
AND 1005.01  ; RK_05 U2_Y #2入壳Y轴滚轮压紧位设定确认
MOVL(498) E1_160 E1_1522  ; RK_05 U2_Y #2入壳Y轴轴当前位置, RK_05 U2_Y #2入壳Y轴滚轮压紧位
LD TR0
AND 1005.02  ; RK_05 U2_Y #2入壳Y轴滚轮松开位设定确认
MOVL(498) E1_160 E1_1524  ; RK_05 U2_Y #2入壳Y轴轴当前位置, RK_05 U2_Y #2入壳Y轴滚轮松开位
LD TR0
AND 1005.03  ; RK_05 U2_Y #2入壳Y轴入壳位设定确认
MOVL(498) E1_160 E1_1526  ; RK_05 U2_Y #2入壳Y轴轴当前位置, RK_05 U2_Y #2入壳Y轴入壳位
LD TR0
AND 1005.04  ; RK_05 U2_Y #2入壳Y轴电芯定位夹爪松开位设定确认
MOVL(498) E1_160 E1_1528  ; RK_05 U2_Y #2入壳Y轴轴当前位置, RK_05 U2_Y #2入壳Y轴电芯定位夹爪松开位
; rung 38: RK_05 U2_Y #2入壳Y轴运行条件
LDNOT 802.10  ; RK_05 U2_Y #2入壳Y轴报警信号标志[0002.10]
AND 802.11  ; RK_05 U2_Y #2入壳Y轴准备好了信号标志[0002.11]
ANDNOT 200.01  ; 紧急停止
ANDNOT 2022.15  ; RK_05 U2_Y #2入壳Y轴停止
OUT D1062.00  ; RK_05 U2_Y #2入壳Y轴运行条件
; rung 39: RK_05 U2_Y #2入壳Y轴回原点条件
LD 804.13  ; RK_05 #2入壳电芯#1定位夹爪气缸松开位标志[0004.13]
AND 804.14  ; RK_05 #2入壳电芯#2定位夹爪气缸松开位标志[0004.14]
LD H20.00  ; RK_03 U0_U 电芯上料X轴回原点记忆
ANDNOT 853.03  ; RK_03 U0_U 电芯上料X轴#2入壳放料位标志
OR 800.09  ; RK_03 电芯上料升降气缸上升位标志[0000.09]
ANDLD
OUT D1062.01  ; RK_05 U2_Y #2入壳Y轴回原点条件

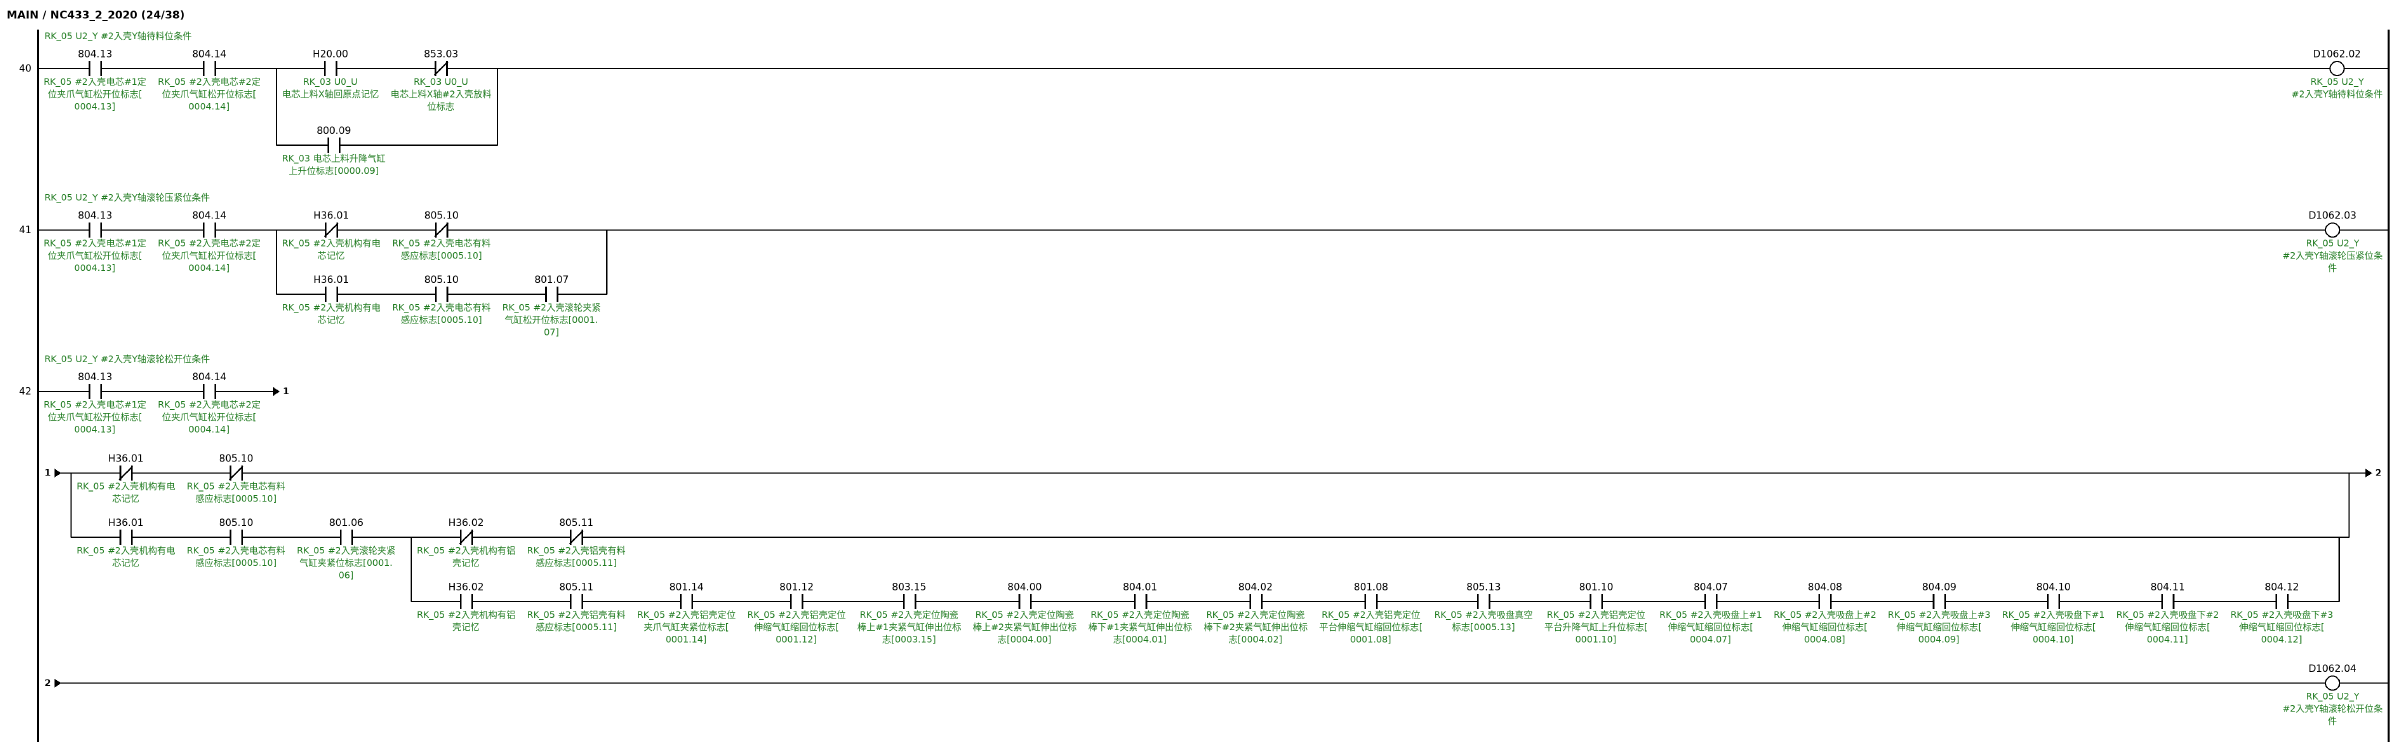
; rung 40: RK_05 U2_Y #2入壳Y轴待料位条件
LD 804.13  ; RK_05 #2入壳电芯#1定位夹爪气缸松开位标志[0004.13]
AND 804.14  ; RK_05 #2入壳电芯#2定位夹爪气缸松开位标志[0004.14]
LD H20.00  ; RK_03 U0_U 电芯上料X轴回原点记忆
ANDNOT 853.03  ; RK_03 U0_U 电芯上料X轴#2入壳放料位标志
OR 800.09  ; RK_03 电芯上料升降气缸上升位标志[0000.09]
ANDLD
OUT D1062.02  ; RK_05 U2_Y #2入壳Y轴待料位条件
; rung 41: RK_05 U2_Y #2入壳Y轴滚轮压紧位条件
LD 804.13  ; RK_05 #2入壳电芯#1定位夹爪气缸松开位标志[0004.13]
AND 804.14  ; RK_05 #2入壳电芯#2定位夹爪气缸松开位标志[0004.14]
LDNOT H36.01  ; RK_05 #2入壳机构有电芯记忆
ANDNOT 805.10  ; RK_05 #2入壳电芯有料感应标志[0005.10]
LD H36.01  ; RK_05 #2入壳机构有电芯记忆
AND 805.10  ; RK_05 #2入壳电芯有料感应标志[0005.10]
AND 801.07  ; RK_05 #2入壳滚轮夹紧气缸松开位标志[0001.07]
ORLD
ANDLD
OUT D1062.03  ; RK_05 U2_Y #2入壳Y轴滚轮压紧位条件
; rung 42: RK_05 U2_Y #2入壳Y轴滚轮松开位条件
LD 804.13  ; RK_05 #2入壳电芯#1定位夹爪气缸松开位标志[0004.13]
AND 804.14  ; RK_05 #2入壳电芯#2定位夹爪气缸松开位标志[0004.14]
LDNOT H36.01  ; RK_05 #2入壳机构有电芯记忆
ANDNOT 805.10  ; RK_05 #2入壳电芯有料感应标志[0005.10]
LD H36.01  ; RK_05 #2入壳机构有电芯记忆
AND 805.10  ; RK_05 #2入壳电芯有料感应标志[0005.10]
AND 801.06  ; RK_05 #2入壳滚轮夹紧气缸夹紧位标志[0001.06]
LDNOT H36.02  ; RK_05 #2入壳机构有铝壳记忆
ANDNOT 805.11  ; RK_05 #2入壳铝壳有料感应标志[0005.11]
LD H36.02  ; RK_05 #2入壳机构有铝壳记忆
AND 805.11  ; RK_05 #2入壳铝壳有料感应标志[0005.11]
AND 801.14  ; RK_05 #2入壳铝壳定位夹爪气缸夹紧位标志[0001.14]
AND 801.12  ; RK_05 #2入壳铝壳定位伸缩气缸缩回位标志[0001.12]
AND 803.15  ; RK_05 #2入壳定位陶瓷棒上#1夹紧气缸伸出位标志[0003.15]
AND 804.00  ; RK_05 #2入壳定位陶瓷棒上#2夹紧气缸伸出位标志[0004.00]
AND 804.01  ; RK_05 #2入壳定位陶瓷棒下#1夹紧气缸伸出位标志[0004.01]
AND 804.02  ; RK_05 #2入壳定位陶瓷棒下#2夹紧气缸伸出位标志[0004.02]
AND 801.08  ; RK_05 #2入壳铝壳定位平台伸缩气缸缩回位标志[0001.08]
AND 805.13  ; RK_05 #2入壳吸盘真空标志[0005.13]
AND 801.10  ; RK_05 #2入壳铝壳定位平台升降气缸上升位标志[0001.10]
AND 804.07  ; RK_05 #2入壳吸盘上#1伸缩气缸缩回位标志[0004.07]
AND 804.08  ; RK_05 #2入壳吸盘上#2伸缩气缸缩回位标志[0004.08]
AND 804.09  ; RK_05 #2入壳吸盘上#3伸缩气缸缩回位标志[0004.09]
AND 804.10  ; RK_05 #2入壳吸盘下#1伸缩气缸缩回位标志[0004.10]
AND 804.11  ; RK_05 #2入壳吸盘下#2伸缩气缸缩回位标志[0004.11]
AND 804.12  ; RK_05 #2入壳吸盘下#3伸缩气缸缩回位标志[0004.12]
ORLD
ANDLD
ORLD
ANDLD
OUT D1062.04  ; RK_05 U2_Y #2入壳Y轴滚轮松开位条件

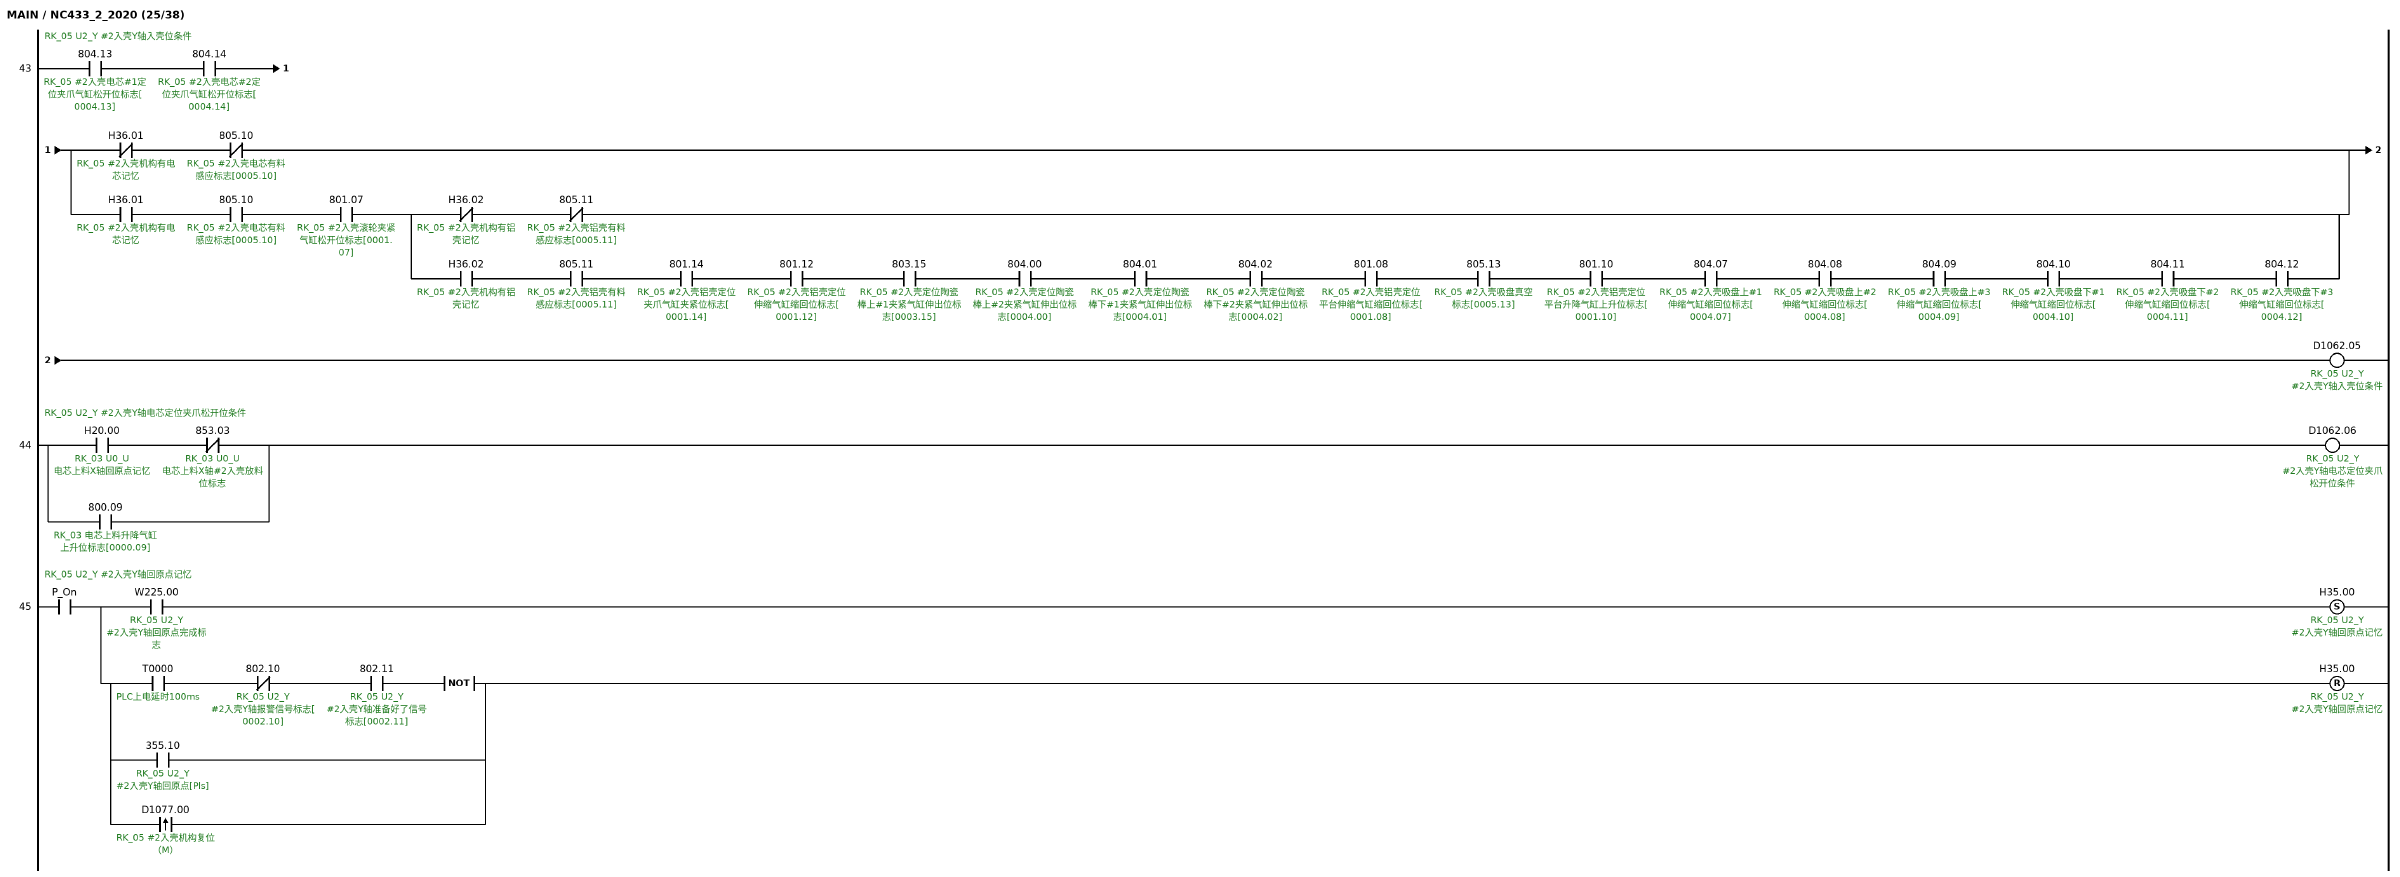
; rung 43: RK_05 U2_Y #2入壳Y轴入壳位条件
LD 804.13  ; RK_05 #2入壳电芯#1定位夹爪气缸松开位标志[0004.13]
AND 804.14  ; RK_05 #2入壳电芯#2定位夹爪气缸松开位标志[0004.14]
LDNOT H36.01  ; RK_05 #2入壳机构有电芯记忆
ANDNOT 805.10  ; RK_05 #2入壳电芯有料感应标志[0005.10]
LD H36.01  ; RK_05 #2入壳机构有电芯记忆
AND 805.10  ; RK_05 #2入壳电芯有料感应标志[0005.10]
AND 801.07  ; RK_05 #2入壳滚轮夹紧气缸松开位标志[0001.07]
LDNOT H36.02  ; RK_05 #2入壳机构有铝壳记忆
ANDNOT 805.11  ; RK_05 #2入壳铝壳有料感应标志[0005.11]
LD H36.02  ; RK_05 #2入壳机构有铝壳记忆
AND 805.11  ; RK_05 #2入壳铝壳有料感应标志[0005.11]
AND 801.14  ; RK_05 #2入壳铝壳定位夹爪气缸夹紧位标志[0001.14]
AND 801.12  ; RK_05 #2入壳铝壳定位伸缩气缸缩回位标志[0001.12]
AND 803.15  ; RK_05 #2入壳定位陶瓷棒上#1夹紧气缸伸出位标志[0003.15]
AND 804.00  ; RK_05 #2入壳定位陶瓷棒上#2夹紧气缸伸出位标志[0004.00]
AND 804.01  ; RK_05 #2入壳定位陶瓷棒下#1夹紧气缸伸出位标志[0004.01]
AND 804.02  ; RK_05 #2入壳定位陶瓷棒下#2夹紧气缸伸出位标志[0004.02]
AND 801.08  ; RK_05 #2入壳铝壳定位平台伸缩气缸缩回位标志[0001.08]
AND 805.13  ; RK_05 #2入壳吸盘真空标志[0005.13]
AND 801.10  ; RK_05 #2入壳铝壳定位平台升降气缸上升位标志[0001.10]
AND 804.07  ; RK_05 #2入壳吸盘上#1伸缩气缸缩回位标志[0004.07]
AND 804.08  ; RK_05 #2入壳吸盘上#2伸缩气缸缩回位标志[0004.08]
AND 804.09  ; RK_05 #2入壳吸盘上#3伸缩气缸缩回位标志[0004.09]
AND 804.10  ; RK_05 #2入壳吸盘下#1伸缩气缸缩回位标志[0004.10]
AND 804.11  ; RK_05 #2入壳吸盘下#2伸缩气缸缩回位标志[0004.11]
AND 804.12  ; RK_05 #2入壳吸盘下#3伸缩气缸缩回位标志[0004.12]
ORLD
ANDLD
ORLD
ANDLD
OUT D1062.05  ; RK_05 U2_Y #2入壳Y轴入壳位条件
; rung 44: RK_05 U2_Y #2入壳Y轴电芯定位夹爪松开位条件
LD H20.00  ; RK_03 U0_U 电芯上料X轴回原点记忆
ANDNOT 853.03  ; RK_03 U0_U 电芯上料X轴#2入壳放料位标志
OR 800.09  ; RK_03 电芯上料升降气缸上升位标志[0000.09]
OUT D1062.06  ; RK_05 U2_Y #2入壳Y轴电芯定位夹爪松开位条件
; rung 45: RK_05 U2_Y #2入壳Y轴回原点记忆
LD P_On
OUT TR0
AND W225.00  ; RK_05 U2_Y #2入壳Y轴回原点完成标志
SET H35.00  ; RK_05 U2_Y #2入壳Y轴回原点记忆
LD TR0
LD T0000  ; PLC上电延时100ms
ANDNOT 802.10  ; RK_05 U2_Y #2入壳Y轴报警信号标志[0002.10]
AND 802.11  ; RK_05 U2_Y #2入壳Y轴准备好了信号标志[0002.11]
NOT(520)
OR 355.10  ; RK_05 U2_Y #2入壳Y轴回原点[Pls]
@OR D1077.00  ; RK_05 #2入壳机构复位（M）
ANDLD
RSET H35.00  ; RK_05 U2_Y #2入壳Y轴回原点记忆

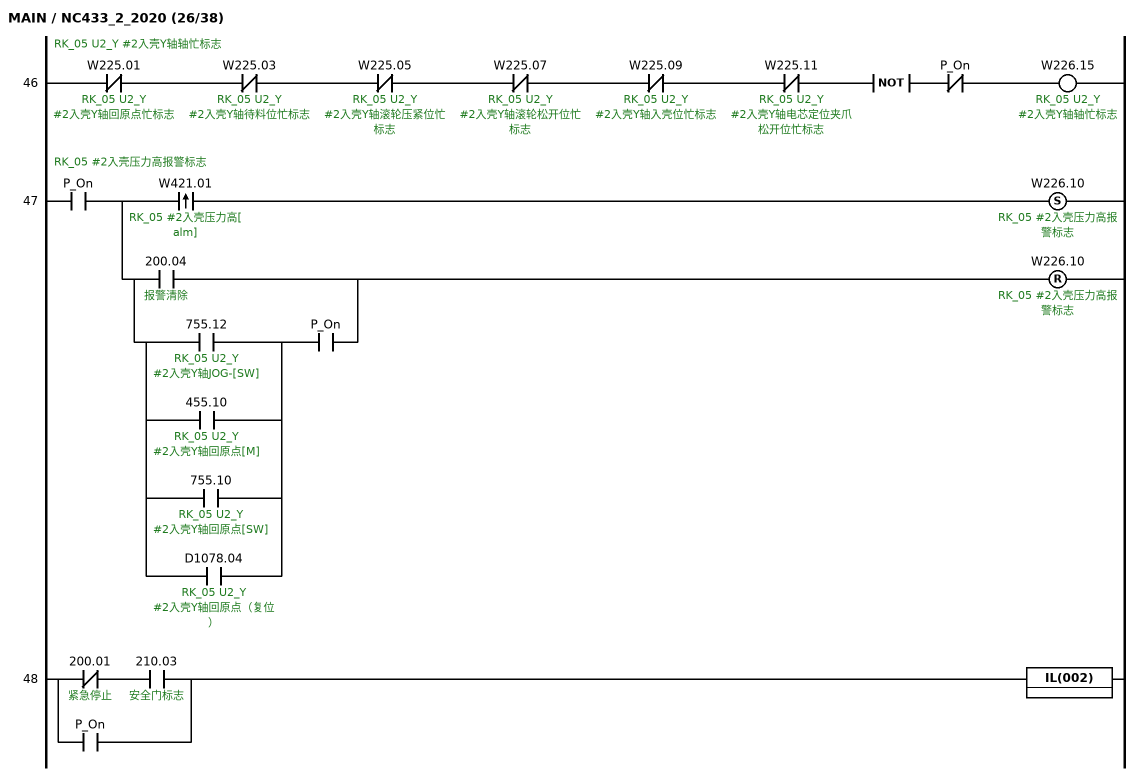
; rung 46: RK_05 U2_Y #2入壳Y轴轴忙标志
LDNOT W225.01  ; RK_05 U2_Y #2入壳Y轴回原点忙标志
ANDNOT W225.03  ; RK_05 U2_Y #2入壳Y轴待料位忙标志
ANDNOT W225.05  ; RK_05 U2_Y #2入壳Y轴滚轮压紧位忙标志
ANDNOT W225.07  ; RK_05 U2_Y #2入壳Y轴滚轮松开位忙标志
ANDNOT W225.09  ; RK_05 U2_Y #2入壳Y轴入壳位忙标志
ANDNOT W225.11  ; RK_05 U2_Y #2入壳Y轴电芯定位夹爪松开位忙标志
NOT(520)
ANDNOT P_On
OUT W226.15  ; RK_05 U2_Y #2入壳Y轴轴忙标志
; rung 47: RK_05 #2入壳压力高报警标志
LD P_On
OUT TR0
@AND W421.01  ; RK_05 #2入壳压力高[alm]
SET W226.10  ; RK_05 #2入壳压力高报警标志
LD TR0
LD 200.04  ; 报警清除
LD 755.12  ; RK_05 U2_Y #2入壳Y轴JOG-[SW]
OR 455.10  ; RK_05 U2_Y #2入壳Y轴回原点[M]
OR 755.10  ; RK_05 U2_Y #2入壳Y轴回原点[SW]
OR D1078.04  ; RK_05 U2_Y #2入壳Y轴回原点（复位）
AND P_On
ORLD
ANDLD
RSET W226.10  ; RK_05 #2入壳压力高报警标志
; rung 48
LDNOT 200.01  ; 紧急停止
AND 210.03  ; 安全门标志
OR P_On
IL(002)

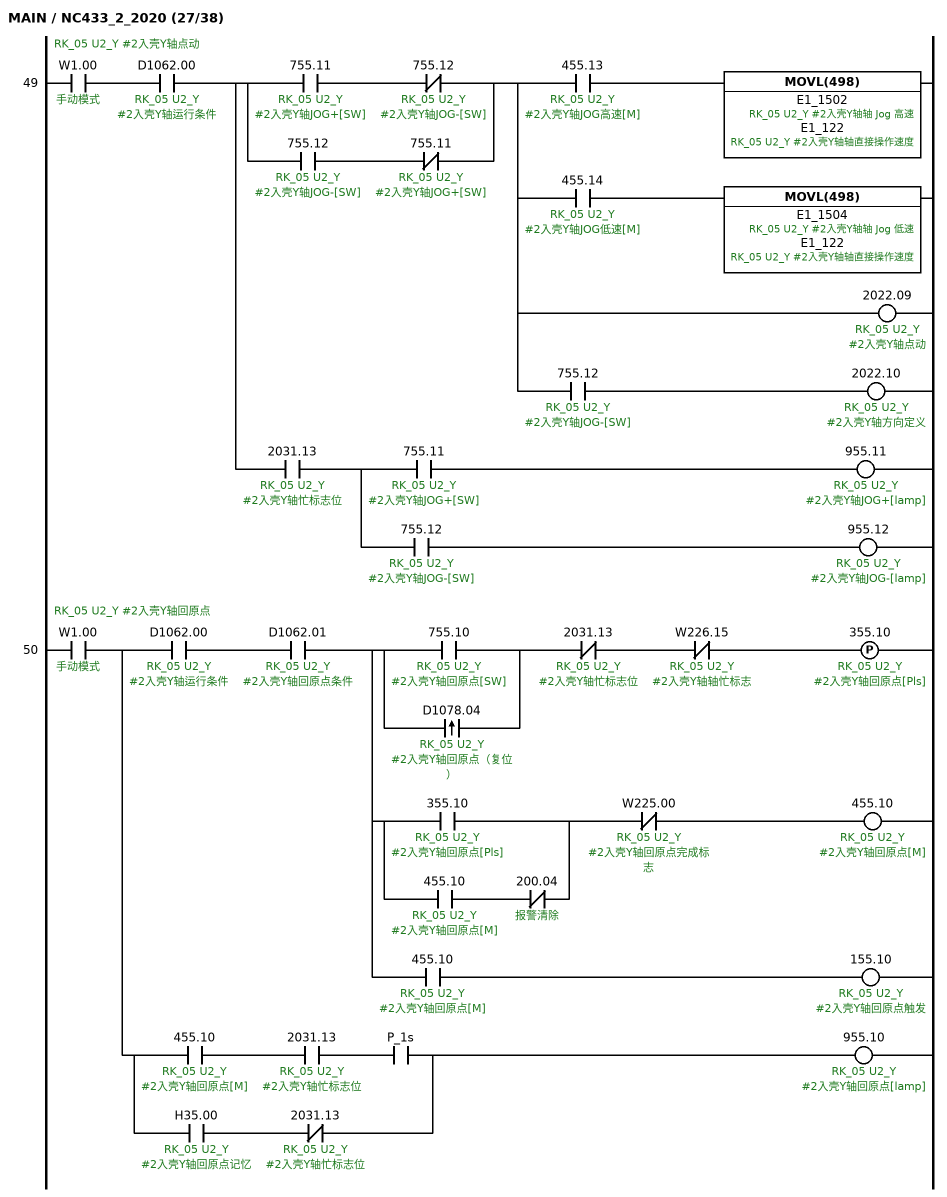
; rung 49: RK_05 U2_Y #2入壳Y轴点动
LD W1.00  ; 手动模式
AND D1062.00  ; RK_05 U2_Y #2入壳Y轴运行条件
OUT TR0
LD 755.11  ; RK_05 U2_Y #2入壳Y轴JOG+[SW]
ANDNOT 755.12  ; RK_05 U2_Y #2入壳Y轴JOG-[SW]
LD 755.12  ; RK_05 U2_Y #2入壳Y轴JOG-[SW]
ANDNOT 755.11  ; RK_05 U2_Y #2入壳Y轴JOG+[SW]
ORLD
ANDLD
OUT TR1
AND 455.13  ; RK_05 U2_Y #2入壳Y轴JOG高速[M]
MOVL(498) E1_1502 E1_122  ; RK_05 U2_Y #2入壳Y轴轴 Jog 高速, RK_05 U2_Y #2入壳Y轴轴直接操作速度
LD TR1
AND 455.14  ; RK_05 U2_Y #2入壳Y轴JOG低速[M]
MOVL(498) E1_1504 E1_122  ; RK_05 U2_Y #2入壳Y轴轴 Jog 低速, RK_05 U2_Y #2入壳Y轴轴直接操作速度
LD TR1
OUT 2022.09  ; RK_05 U2_Y #2入壳Y轴点动
AND 755.12  ; RK_05 U2_Y #2入壳Y轴JOG-[SW]
OUT 2022.10  ; RK_05 U2_Y #2入壳Y轴方向定义
LD TR0
AND 2031.13  ; RK_05 U2_Y #2入壳Y轴忙标志位
OUT TR0
AND 755.11  ; RK_05 U2_Y #2入壳Y轴JOG+[SW]
OUT 955.11  ; RK_05 U2_Y #2入壳Y轴JOG+[lamp]
LD TR0
AND 755.12  ; RK_05 U2_Y #2入壳Y轴JOG-[SW]
OUT 955.12  ; RK_05 U2_Y #2入壳Y轴JOG-[lamp]
; rung 50: RK_05 U2_Y #2入壳Y轴回原点
LD W1.00  ; 手动模式
OUT TR0
AND D1062.00  ; RK_05 U2_Y #2入壳Y轴运行条件
AND D1062.01  ; RK_05 U2_Y #2入壳Y轴回原点条件
OUT TR1
LD 755.10  ; RK_05 U2_Y #2入壳Y轴回原点[SW]
@OR D1078.04  ; RK_05 U2_Y #2入壳Y轴回原点（复位）
ANDLD
ANDNOT 2031.13  ; RK_05 U2_Y #2入壳Y轴忙标志位
ANDNOT W226.15  ; RK_05 U2_Y #2入壳Y轴轴忙标志
DIFU(013) 355.10  ; RK_05 U2_Y #2入壳Y轴回原点[Pls]
LD TR1
LD 355.10  ; RK_05 U2_Y #2入壳Y轴回原点[Pls]
LD 455.10  ; RK_05 U2_Y #2入壳Y轴回原点[M]
ANDNOT 200.04  ; 报警清除
ORLD
ANDLD
ANDNOT W225.00  ; RK_05 U2_Y #2入壳Y轴回原点完成标志
OUT 455.10  ; RK_05 U2_Y #2入壳Y轴回原点[M]
LD TR1
AND 455.10  ; RK_05 U2_Y #2入壳Y轴回原点[M]
OUT 155.10  ; RK_05 U2_Y #2入壳Y轴回原点触发
LD TR0
LD 455.10  ; RK_05 U2_Y #2入壳Y轴回原点[M]
AND 2031.13  ; RK_05 U2_Y #2入壳Y轴忙标志位
AND P_1s
LD H35.00  ; RK_05 U2_Y #2入壳Y轴回原点记忆
ANDNOT 2031.13  ; RK_05 U2_Y #2入壳Y轴忙标志位
ORLD
ANDLD
OUT 955.10  ; RK_05 U2_Y #2入壳Y轴回原点[lamp]

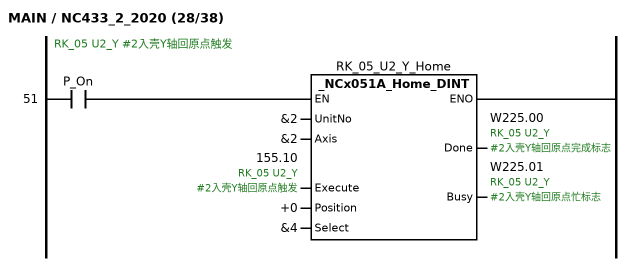
; rung 51: RK_05 U2_Y #2入壳Y轴回原点触发
LD P_On
CALL RK_05_U2_Y_Home : _NCx051A_Home_DINT (UnitNo := &2, Axis := &2, Execute := 155.10, Position := +0, Select := &4, Done => W225.00, Busy => W225.01)  ; RK_05 U2_Y #2入壳Y轴回原点触发, RK_05 U2_Y #2入壳Y轴回原点完成标志, RK_05 U2_Y #2入壳Y轴回原点忙标志

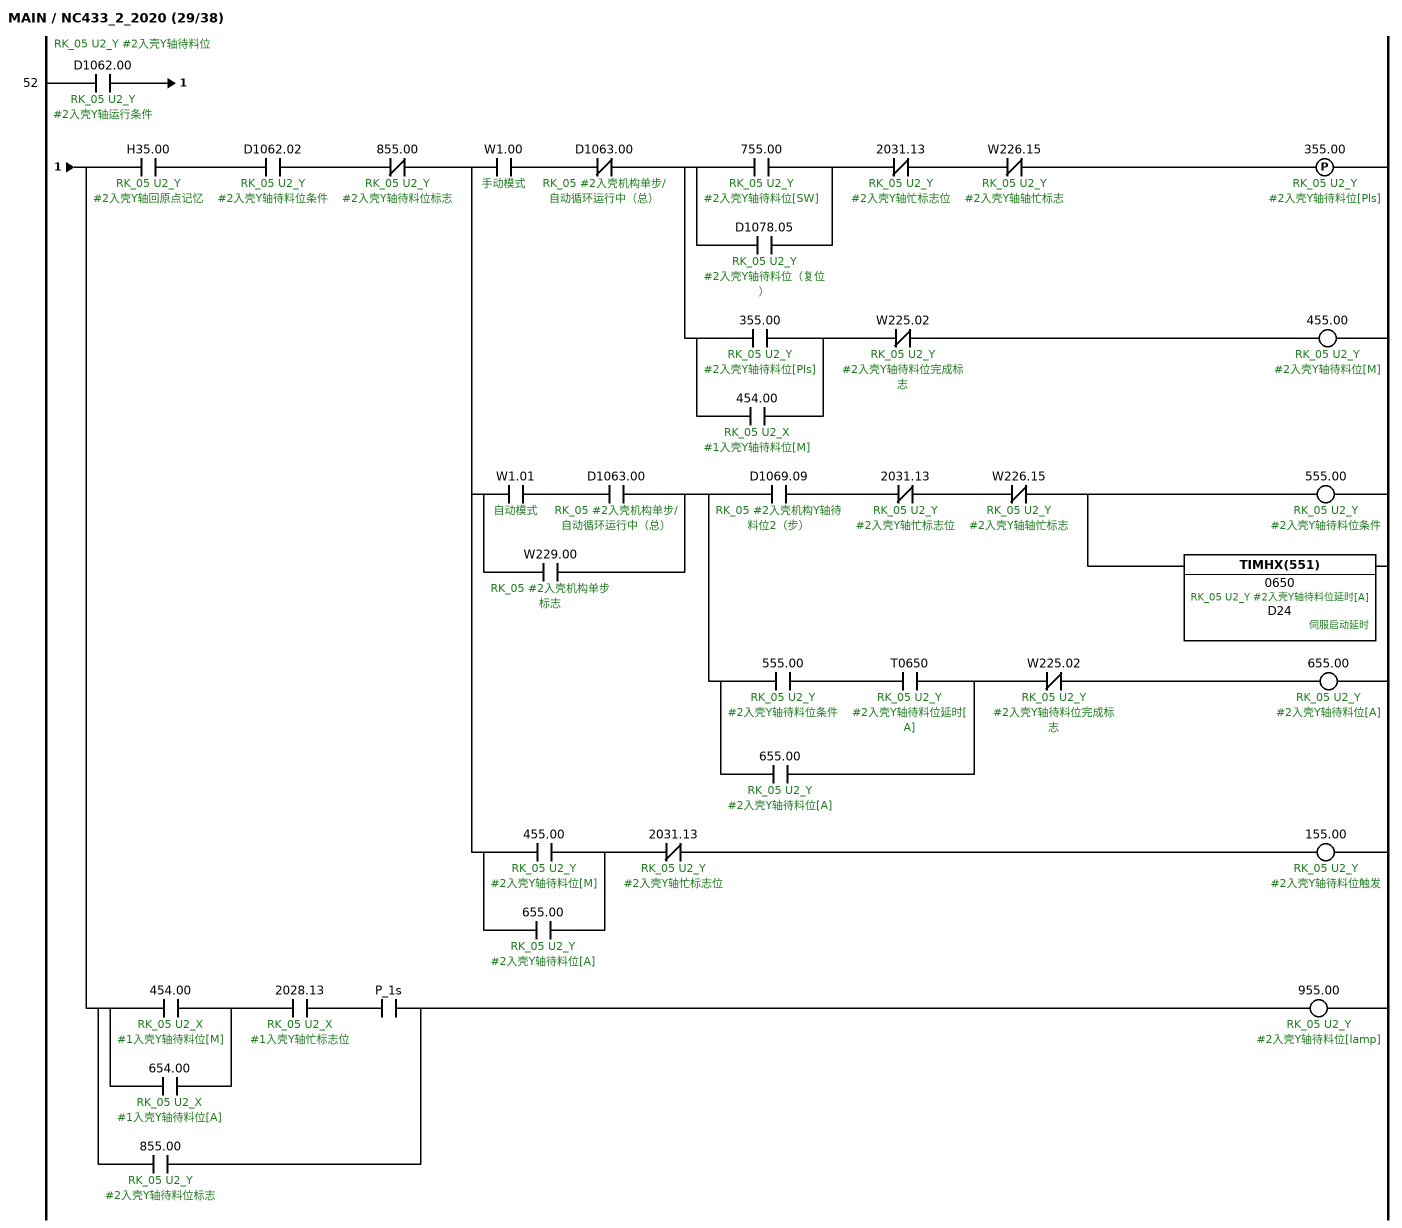
; rung 52: RK_05 U2_Y #2入壳Y轴待料位
LD D1062.00  ; RK_05 U2_Y #2入壳Y轴运行条件
OUT TR0
AND H35.00  ; RK_05 U2_Y #2入壳Y轴回原点记忆
AND D1062.02  ; RK_05 U2_Y #2入壳Y轴待料位条件
ANDNOT 855.00  ; RK_05 U2_Y #2入壳Y轴待料位标志
OUT TR1
AND W1.00  ; 手动模式
ANDNOT D1063.00  ; RK_05 #2入壳机构单步/自动循环运行中（总）
OUT TR2
LD 755.00  ; RK_05 U2_Y #2入壳Y轴待料位[SW]
OR D1078.05  ; RK_05 U2_Y #2入壳Y轴待料位（复位）
ANDLD
ANDNOT 2031.13  ; RK_05 U2_Y #2入壳Y轴忙标志位
ANDNOT W226.15  ; RK_05 U2_Y #2入壳Y轴轴忙标志
DIFU(013) 355.00  ; RK_05 U2_Y #2入壳Y轴待料位[Pls]
LD TR2
LD 355.00  ; RK_05 U2_Y #2入壳Y轴待料位[Pls]
OR 454.00  ; RK_05 U2_X #1入壳Y轴待料位[M]
ANDLD
ANDNOT W225.02  ; RK_05 U2_Y #2入壳Y轴待料位完成标志
OUT 455.00  ; RK_05 U2_Y #2入壳Y轴待料位[M]
LD TR1
LD W1.01  ; 自动模式
AND D1063.00  ; RK_05 #2入壳机构单步/自动循环运行中（总）
OR W229.00  ; RK_05 #2入壳机构单步标志
ANDLD
OUT TR2
AND D1069.09  ; RK_05 #2入壳机构Y轴待料位2（步）
ANDNOT 2031.13  ; RK_05 U2_Y #2入壳Y轴忙标志位
ANDNOT W226.15  ; RK_05 U2_Y #2入壳Y轴轴忙标志
OUT 555.00  ; RK_05 U2_Y #2入壳Y轴待料位条件
TIMHX(551) 0650 D24  ; 伺服启动延时, RK_05 U2_Y #2入壳Y轴待料位延时[A]
LD TR2
LD 555.00  ; RK_05 U2_Y #2入壳Y轴待料位条件
AND T0650  ; RK_05 U2_Y #2入壳Y轴待料位延时[A]
OR 655.00  ; RK_05 U2_Y #2入壳Y轴待料位[A]
ANDLD
ANDNOT W225.02  ; RK_05 U2_Y #2入壳Y轴待料位完成标志
OUT 655.00  ; RK_05 U2_Y #2入壳Y轴待料位[A]
LD TR1
LD 455.00  ; RK_05 U2_Y #2入壳Y轴待料位[M]
OR 655.00  ; RK_05 U2_Y #2入壳Y轴待料位[A]
ANDLD
ANDNOT 2031.13  ; RK_05 U2_Y #2入壳Y轴忙标志位
OUT 155.00  ; RK_05 U2_Y #2入壳Y轴待料位触发
LD TR0
LD 454.00  ; RK_05 U2_X #1入壳Y轴待料位[M]
OR 654.00  ; RK_05 U2_X #1入壳Y轴待料位[A]
AND 2028.13  ; RK_05 U2_X #1入壳Y轴忙标志位
AND P_1s
OR 855.00  ; RK_05 U2_Y #2入壳Y轴待料位标志
ANDLD
OUT 955.00  ; RK_05 U2_Y #2入壳Y轴待料位[lamp]

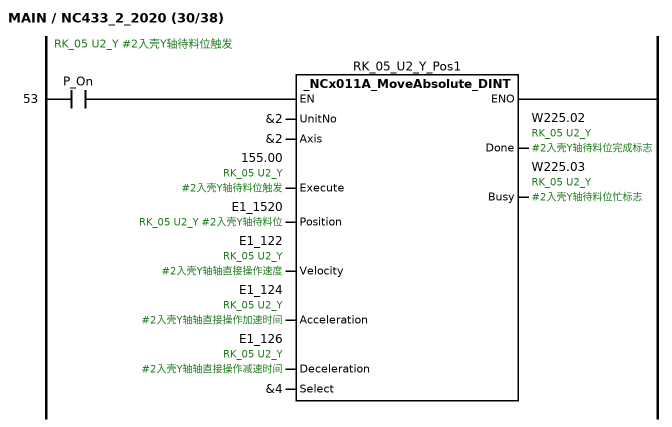
; rung 53: RK_05 U2_Y #2入壳Y轴待料位触发
LD P_On
CALL RK_05_U2_Y_Pos1 : _NCx011A_MoveAbsolute_DINT (UnitNo := &2, Axis := &2, Execute := 155.00, Position := E1_1520, Velocity := E1_122, Acceleration := E1_124, Deceleration := E1_126, Select := &4, Done => W225.02, Busy => W225.03)  ; RK_05 U2_Y #2入壳Y轴待料位触发, RK_05 U2_Y #2入壳Y轴待料位, RK_05 U2_Y #2入壳Y轴轴直接操作速度, RK_05 U2_Y #2入壳Y轴轴直接操作加速时间, RK_05 U2_Y #2入壳Y轴轴直接操作减速时间, RK_05 U2_Y #2入壳Y轴待料位完成标志, RK_05 U2_Y #2入壳Y轴待料位忙标志

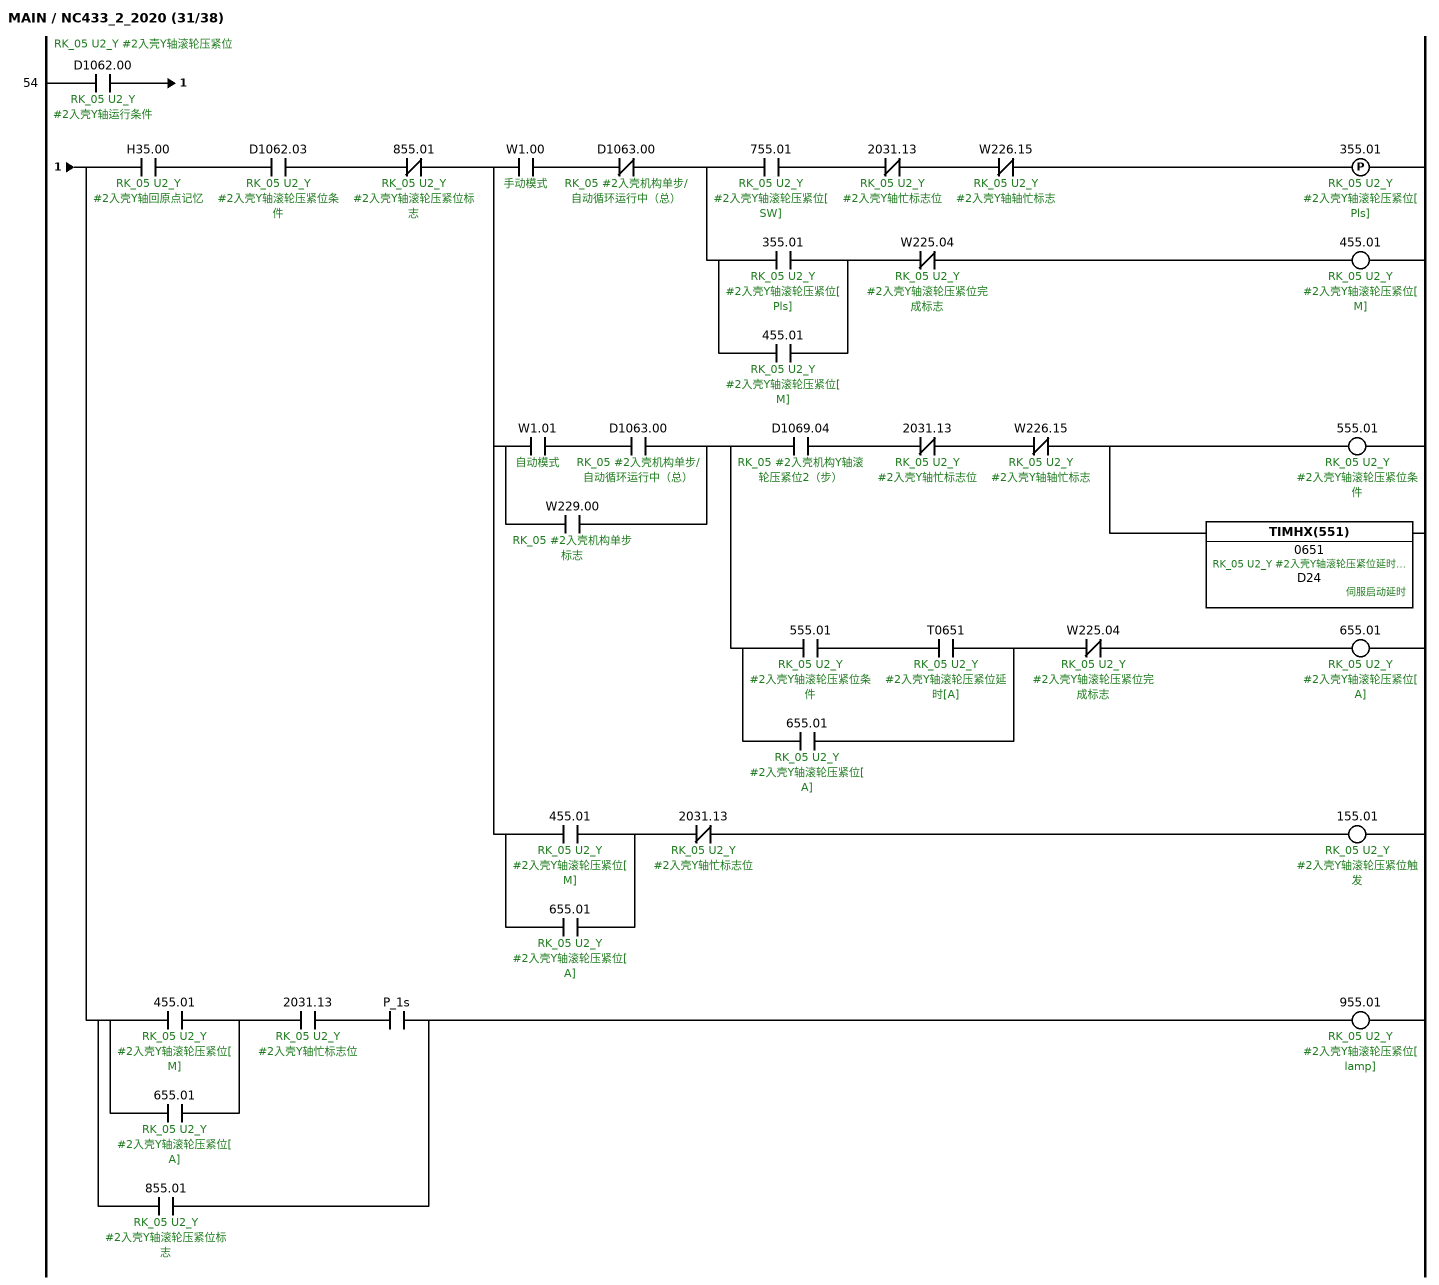
; rung 54: RK_05 U2_Y #2入壳Y轴滚轮压紧位
LD D1062.00  ; RK_05 U2_Y #2入壳Y轴运行条件
OUT TR0
AND H35.00  ; RK_05 U2_Y #2入壳Y轴回原点记忆
AND D1062.03  ; RK_05 U2_Y #2入壳Y轴滚轮压紧位条件
ANDNOT 855.01  ; RK_05 U2_Y #2入壳Y轴滚轮压紧位标志
OUT TR1
AND W1.00  ; 手动模式
ANDNOT D1063.00  ; RK_05 #2入壳机构单步/自动循环运行中（总）
OUT TR2
AND 755.01  ; RK_05 U2_Y #2入壳Y轴滚轮压紧位[SW]
ANDNOT 2031.13  ; RK_05 U2_Y #2入壳Y轴忙标志位
ANDNOT W226.15  ; RK_05 U2_Y #2入壳Y轴轴忙标志
DIFU(013) 355.01  ; RK_05 U2_Y #2入壳Y轴滚轮压紧位[Pls]
LD TR2
LD 355.01  ; RK_05 U2_Y #2入壳Y轴滚轮压紧位[Pls]
OR 455.01  ; RK_05 U2_Y #2入壳Y轴滚轮压紧位[M]
ANDLD
ANDNOT W225.04  ; RK_05 U2_Y #2入壳Y轴滚轮压紧位完成标志
OUT 455.01  ; RK_05 U2_Y #2入壳Y轴滚轮压紧位[M]
LD TR1
LD W1.01  ; 自动模式
AND D1063.00  ; RK_05 #2入壳机构单步/自动循环运行中（总）
OR W229.00  ; RK_05 #2入壳机构单步标志
ANDLD
OUT TR2
AND D1069.04  ; RK_05 #2入壳机构Y轴滚轮压紧位2（步）
ANDNOT 2031.13  ; RK_05 U2_Y #2入壳Y轴忙标志位
ANDNOT W226.15  ; RK_05 U2_Y #2入壳Y轴轴忙标志
OUT 555.01  ; RK_05 U2_Y #2入壳Y轴滚轮压紧位条件
TIMHX(551) 0651 D24  ; 伺服启动延时, RK_05 U2_Y #2入壳Y轴滚轮压紧位延时[A]
LD TR2
LD 555.01  ; RK_05 U2_Y #2入壳Y轴滚轮压紧位条件
AND T0651  ; RK_05 U2_Y #2入壳Y轴滚轮压紧位延时[A]
OR 655.01  ; RK_05 U2_Y #2入壳Y轴滚轮压紧位[A]
ANDLD
ANDNOT W225.04  ; RK_05 U2_Y #2入壳Y轴滚轮压紧位完成标志
OUT 655.01  ; RK_05 U2_Y #2入壳Y轴滚轮压紧位[A]
LD TR1
LD 455.01  ; RK_05 U2_Y #2入壳Y轴滚轮压紧位[M]
OR 655.01  ; RK_05 U2_Y #2入壳Y轴滚轮压紧位[A]
ANDLD
ANDNOT 2031.13  ; RK_05 U2_Y #2入壳Y轴忙标志位
OUT 155.01  ; RK_05 U2_Y #2入壳Y轴滚轮压紧位触发
LD TR0
LD 455.01  ; RK_05 U2_Y #2入壳Y轴滚轮压紧位[M]
OR 655.01  ; RK_05 U2_Y #2入壳Y轴滚轮压紧位[A]
AND 2031.13  ; RK_05 U2_Y #2入壳Y轴忙标志位
AND P_1s
OR 855.01  ; RK_05 U2_Y #2入壳Y轴滚轮压紧位标志
ANDLD
OUT 955.01  ; RK_05 U2_Y #2入壳Y轴滚轮压紧位[lamp]

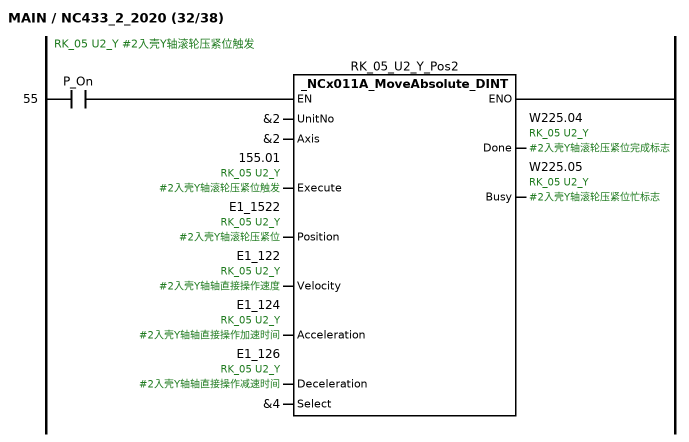
; rung 55: RK_05 U2_Y #2入壳Y轴滚轮压紧位触发
LD P_On
CALL RK_05_U2_Y_Pos2 : _NCx011A_MoveAbsolute_DINT (UnitNo := &2, Axis := &2, Execute := 155.01, Position := E1_1522, Velocity := E1_122, Acceleration := E1_124, Deceleration := E1_126, Select := &4, Done => W225.04, Busy => W225.05)  ; RK_05 U2_Y #2入壳Y轴滚轮压紧位触发, RK_05 U2_Y #2入壳Y轴滚轮压紧位, RK_05 U2_Y #2入壳Y轴轴直接操作速度, RK_05 U2_Y #2入壳Y轴轴直接操作加速时间, RK_05 U2_Y #2入壳Y轴轴直接操作减速时间, RK_05 U2_Y #2入壳Y轴滚轮压紧位完成标志, RK_05 U2_Y #2入壳Y轴滚轮压紧位忙标志

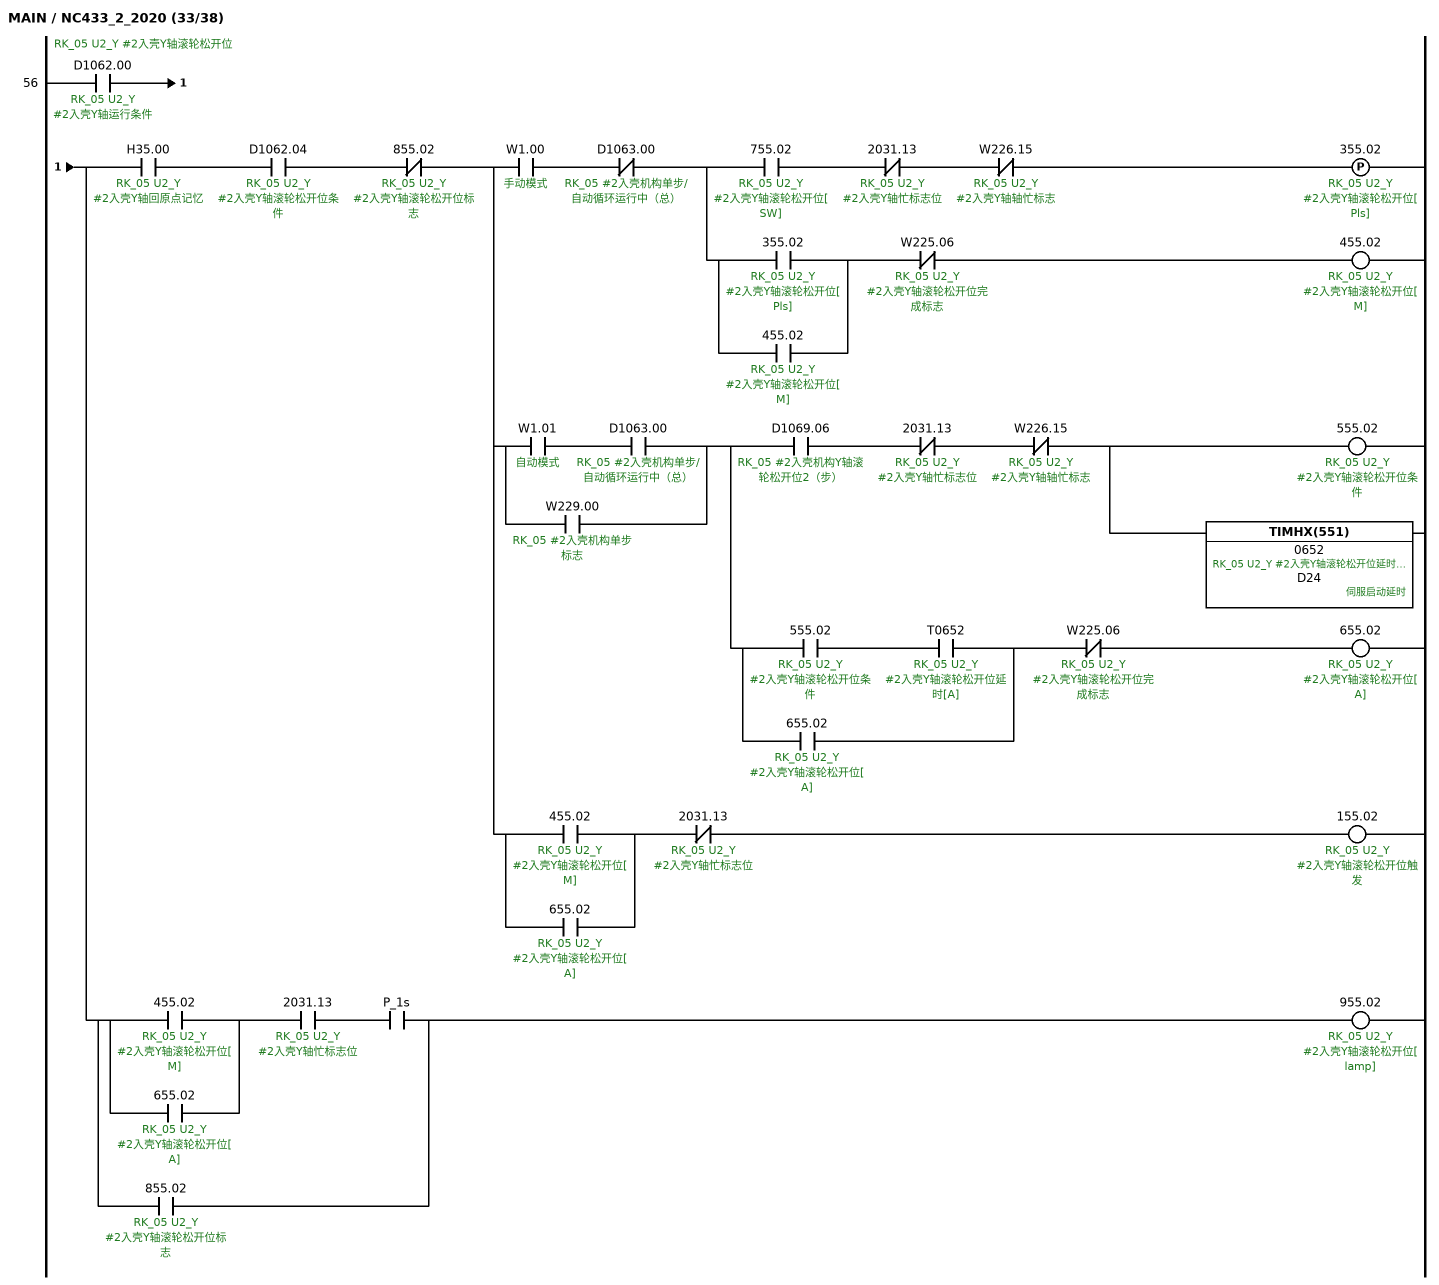
; rung 56: RK_05 U2_Y #2入壳Y轴滚轮松开位
LD D1062.00  ; RK_05 U2_Y #2入壳Y轴运行条件
OUT TR0
AND H35.00  ; RK_05 U2_Y #2入壳Y轴回原点记忆
AND D1062.04  ; RK_05 U2_Y #2入壳Y轴滚轮松开位条件
ANDNOT 855.02  ; RK_05 U2_Y #2入壳Y轴滚轮松开位标志
OUT TR1
AND W1.00  ; 手动模式
ANDNOT D1063.00  ; RK_05 #2入壳机构单步/自动循环运行中（总）
OUT TR2
AND 755.02  ; RK_05 U2_Y #2入壳Y轴滚轮松开位[SW]
ANDNOT 2031.13  ; RK_05 U2_Y #2入壳Y轴忙标志位
ANDNOT W226.15  ; RK_05 U2_Y #2入壳Y轴轴忙标志
DIFU(013) 355.02  ; RK_05 U2_Y #2入壳Y轴滚轮松开位[Pls]
LD TR2
LD 355.02  ; RK_05 U2_Y #2入壳Y轴滚轮松开位[Pls]
OR 455.02  ; RK_05 U2_Y #2入壳Y轴滚轮松开位[M]
ANDLD
ANDNOT W225.06  ; RK_05 U2_Y #2入壳Y轴滚轮松开位完成标志
OUT 455.02  ; RK_05 U2_Y #2入壳Y轴滚轮松开位[M]
LD TR1
LD W1.01  ; 自动模式
AND D1063.00  ; RK_05 #2入壳机构单步/自动循环运行中（总）
OR W229.00  ; RK_05 #2入壳机构单步标志
ANDLD
OUT TR2
AND D1069.06  ; RK_05 #2入壳机构Y轴滚轮松开位2（步）
ANDNOT 2031.13  ; RK_05 U2_Y #2入壳Y轴忙标志位
ANDNOT W226.15  ; RK_05 U2_Y #2入壳Y轴轴忙标志
OUT 555.02  ; RK_05 U2_Y #2入壳Y轴滚轮松开位条件
TIMHX(551) 0652 D24  ; 伺服启动延时, RK_05 U2_Y #2入壳Y轴滚轮松开位延时[A]
LD TR2
LD 555.02  ; RK_05 U2_Y #2入壳Y轴滚轮松开位条件
AND T0652  ; RK_05 U2_Y #2入壳Y轴滚轮松开位延时[A]
OR 655.02  ; RK_05 U2_Y #2入壳Y轴滚轮松开位[A]
ANDLD
ANDNOT W225.06  ; RK_05 U2_Y #2入壳Y轴滚轮松开位完成标志
OUT 655.02  ; RK_05 U2_Y #2入壳Y轴滚轮松开位[A]
LD TR1
LD 455.02  ; RK_05 U2_Y #2入壳Y轴滚轮松开位[M]
OR 655.02  ; RK_05 U2_Y #2入壳Y轴滚轮松开位[A]
ANDLD
ANDNOT 2031.13  ; RK_05 U2_Y #2入壳Y轴忙标志位
OUT 155.02  ; RK_05 U2_Y #2入壳Y轴滚轮松开位触发
LD TR0
LD 455.02  ; RK_05 U2_Y #2入壳Y轴滚轮松开位[M]
OR 655.02  ; RK_05 U2_Y #2入壳Y轴滚轮松开位[A]
AND 2031.13  ; RK_05 U2_Y #2入壳Y轴忙标志位
AND P_1s
OR 855.02  ; RK_05 U2_Y #2入壳Y轴滚轮松开位标志
ANDLD
OUT 955.02  ; RK_05 U2_Y #2入壳Y轴滚轮松开位[lamp]

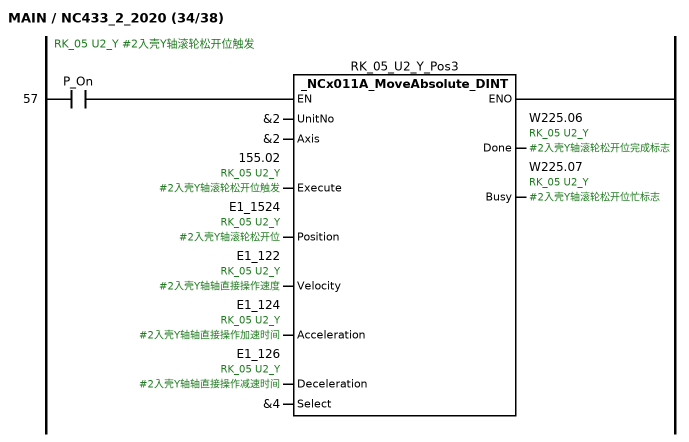
; rung 57: RK_05 U2_Y #2入壳Y轴滚轮松开位触发
LD P_On
CALL RK_05_U2_Y_Pos3 : _NCx011A_MoveAbsolute_DINT (UnitNo := &2, Axis := &2, Execute := 155.02, Position := E1_1524, Velocity := E1_122, Acceleration := E1_124, Deceleration := E1_126, Select := &4, Done => W225.06, Busy => W225.07)  ; RK_05 U2_Y #2入壳Y轴滚轮松开位触发, RK_05 U2_Y #2入壳Y轴滚轮松开位, RK_05 U2_Y #2入壳Y轴轴直接操作速度, RK_05 U2_Y #2入壳Y轴轴直接操作加速时间, RK_05 U2_Y #2入壳Y轴轴直接操作减速时间, RK_05 U2_Y #2入壳Y轴滚轮松开位完成标志, RK_05 U2_Y #2入壳Y轴滚轮松开位忙标志

